    stLENS2_428[0].fEnergy := 8280.000000; stLENS2_428[0].fLow := 51.070000; stLENS2_428[0].fHigh := 10000.000000;
    stLENS2_428[1].fEnergy := 8291.222140; stLENS2_428[1].fLow := 50.858061; stLENS2_428[1].fHigh := 10000.000000;
    stLENS2_428[2].fEnergy := 8307.821178; stLENS2_428[2].fLow := 50.642862; stLENS2_428[2].fHigh := 10000.000000;
    stLENS2_428[3].fEnergy := 8324.453447; stLENS2_428[3].fLow := 50.428659; stLENS2_428[3].fHigh := 10000.000000;
    stLENS2_428[4].fEnergy := 8341.119014; stLENS2_428[4].fLow := 50.215449; stLENS2_428[4].fHigh := 10000.000000;
    stLENS2_428[5].fEnergy := 8357.817945; stLENS2_428[5].fLow := 50.003226; stLENS2_428[5].fHigh := 10000.000000;
    stLENS2_428[6].fEnergy := 8374.550308; stLENS2_428[6].fLow := 49.791984; stLENS2_428[6].fHigh := 10000.000000;
    stLENS2_428[7].fEnergy := 8391.316169; stLENS2_428[7].fLow := 49.581721; stLENS2_428[7].fHigh := 10000.000000;
    stLENS2_428[8].fEnergy := 8408.115595; stLENS2_428[8].fLow := 49.372429; stLENS2_428[8].fHigh := 10000.000000;
    stLENS2_428[9].fEnergy := 8424.948653; stLENS2_428[9].fLow := 49.164106; stLENS2_428[9].fHigh := 10000.000000;
    stLENS2_428[10].fEnergy := 8441.815412; stLENS2_428[10].fLow := 48.956745; stLENS2_428[10].fHigh := 10000.000000;
    stLENS2_428[11].fEnergy := 8458.715938; stLENS2_428[11].fLow := 48.750343; stLENS2_428[11].fHigh := 10000.000000;
    stLENS2_428[12].fEnergy := 8475.650298; stLENS2_428[12].fLow := 48.544894; stLENS2_428[12].fHigh := 10000.000000;
    stLENS2_428[13].fEnergy := 8492.618561; stLENS2_428[13].fLow := 48.340393; stLENS2_428[13].fHigh := 10000.000000;
    stLENS2_428[14].fEnergy := 8509.620795; stLENS2_428[14].fLow := 48.136837; stLENS2_428[14].fHigh := 10000.000000;
    stLENS2_428[15].fEnergy := 8526.657067; stLENS2_428[15].fLow := 47.934219; stLENS2_428[15].fHigh := 10000.000000;
    stLENS2_428[16].fEnergy := 8543.727446; stLENS2_428[16].fLow := 47.732537; stLENS2_428[16].fHigh := 10000.000000;
    stLENS2_428[17].fEnergy := 8560.832000; stLENS2_428[17].fLow := 47.531784; stLENS2_428[17].fHigh := 10000.000000;
    stLENS2_428[18].fEnergy := 8577.970797; stLENS2_428[18].fLow := 47.331957; stLENS2_428[18].fHigh := 10000.000000;
    stLENS2_428[19].fEnergy := 8595.143906; stLENS2_428[19].fLow := 47.133051; stLENS2_428[19].fHigh := 10000.000000;
    stLENS2_428[20].fEnergy := 8612.351395; stLENS2_428[20].fLow := 46.935061; stLENS2_428[20].fHigh := 10000.000000;
    stLENS2_428[21].fEnergy := 8629.593334; stLENS2_428[21].fLow := 46.737983; stLENS2_428[21].fHigh := 10000.000000;
    stLENS2_428[22].fEnergy := 8646.869792; stLENS2_428[22].fLow := 46.541812; stLENS2_428[22].fHigh := 10000.000000;
    stLENS2_428[23].fEnergy := 8664.180837; stLENS2_428[23].fLow := 46.346544; stLENS2_428[23].fHigh := 10000.000000;
    stLENS2_428[24].fEnergy := 8681.526538; stLENS2_428[24].fLow := 46.152174; stLENS2_428[24].fHigh := 10000.000000;
    stLENS2_428[25].fEnergy := 8698.906966; stLENS2_428[25].fLow := 45.958699; stLENS2_428[25].fHigh := 10000.000000;
    stLENS2_428[26].fEnergy := 8716.322189; stLENS2_428[26].fLow := 45.766112; stLENS2_428[26].fHigh := 10000.000000;
    stLENS2_428[27].fEnergy := 8733.772278; stLENS2_428[27].fLow := 45.574411; stLENS2_428[27].fHigh := 10000.000000;
    stLENS2_428[28].fEnergy := 8751.257302; stLENS2_428[28].fLow := 45.383591; stLENS2_428[28].fHigh := 10000.000000;
    stLENS2_428[29].fEnergy := 8768.777330; stLENS2_428[29].fLow := 45.193647; stLENS2_428[29].fHigh := 10000.000000;
    stLENS2_428[30].fEnergy := 8786.332434; stLENS2_428[30].fLow := 45.004575; stLENS2_428[30].fHigh := 10000.000000;
    stLENS2_428[31].fEnergy := 8803.922684; stLENS2_428[31].fLow := 44.816371; stLENS2_428[31].fHigh := 10000.000000;
    stLENS2_428[32].fEnergy := 8821.548149; stLENS2_428[32].fLow := 44.629030; stLENS2_428[32].fHigh := 10000.000000;
    stLENS2_428[33].fEnergy := 8839.208900; stLENS2_428[33].fLow := 44.442549; stLENS2_428[33].fHigh := 10000.000000;
    stLENS2_428[34].fEnergy := 8856.905008; stLENS2_428[34].fLow := 44.256922; stLENS2_428[34].fHigh := 10000.000000;
    stLENS2_428[35].fEnergy := 8874.636543; stLENS2_428[35].fLow := 44.072147; stLENS2_428[35].fHigh := 10000.000000;
    stLENS2_428[36].fEnergy := 8892.403578; stLENS2_428[36].fLow := 43.888218; stLENS2_428[36].fHigh := 10000.000000;
    stLENS2_428[37].fEnergy := 8910.206181; stLENS2_428[37].fLow := 43.705132; stLENS2_428[37].fHigh := 10000.000000;
    stLENS2_428[38].fEnergy := 8928.044426; stLENS2_428[38].fLow := 43.522884; stLENS2_428[38].fHigh := 10000.000000;
    stLENS2_428[39].fEnergy := 8945.918383; stLENS2_428[39].fLow := 43.341470; stLENS2_428[39].fHigh := 10000.000000;
    stLENS2_428[40].fEnergy := 8963.828123; stLENS2_428[40].fLow := 43.160887; stLENS2_428[40].fHigh := 10000.000000;
    stLENS2_428[41].fEnergy := 8981.773719; stLENS2_428[41].fLow := 42.981129; stLENS2_428[41].fHigh := 10000.000000;
    stLENS2_428[42].fEnergy := 8999.755242; stLENS2_428[42].fLow := 42.802194; stLENS2_428[42].fHigh := 10000.000000;
    stLENS2_428[43].fEnergy := 9017.772764; stLENS2_428[43].fLow := 42.624076; stLENS2_428[43].fHigh := 10000.000000;
    stLENS2_428[44].fEnergy := 9035.826357; stLENS2_428[44].fLow := 42.446773; stLENS2_428[44].fHigh := 10000.000000;
    stLENS2_428[45].fEnergy := 9053.916094; stLENS2_428[45].fLow := 42.270279; stLENS2_428[45].fHigh := 10000.000000;
    stLENS2_428[46].fEnergy := 9072.042046; stLENS2_428[46].fLow := 42.094591; stLENS2_428[46].fHigh := 10000.000000;
    stLENS2_428[47].fEnergy := 9090.204286; stLENS2_428[47].fLow := 41.919706; stLENS2_428[47].fHigh := 10000.000000;
    stLENS2_428[48].fEnergy := 9108.402887; stLENS2_428[48].fLow := 41.745618; stLENS2_428[48].fHigh := 10000.000000;
    stLENS2_428[49].fEnergy := 9126.637922; stLENS2_428[49].fLow := 41.572325; stLENS2_428[49].fHigh := 10000.000000;
    stLENS2_428[50].fEnergy := 9144.909463; stLENS2_428[50].fLow := 41.399822; stLENS2_428[50].fHigh := 10000.000000;
    stLENS2_428[51].fEnergy := 9163.217584; stLENS2_428[51].fLow := 41.228106; stLENS2_428[51].fHigh := 10000.000000;
    stLENS2_428[52].fEnergy := 9181.562358; stLENS2_428[52].fLow := 41.057172; stLENS2_428[52].fHigh := 10000.000000;
    stLENS2_428[53].fEnergy := 9199.943858; stLENS2_428[53].fLow := 40.887017; stLENS2_428[53].fHigh := 10000.000000;
    stLENS2_428[54].fEnergy := 9218.362158; stLENS2_428[54].fLow := 40.717637; stLENS2_428[54].fHigh := 10000.000000;
    stLENS2_428[55].fEnergy := 9236.817331; stLENS2_428[55].fLow := 40.549028; stLENS2_428[55].fHigh := 10000.000000;
    stLENS2_428[56].fEnergy := 9255.309452; stLENS2_428[56].fLow := 40.381186; stLENS2_428[56].fHigh := 10000.000000;
    stLENS2_428[57].fEnergy := 9273.838594; stLENS2_428[57].fLow := 40.214108; stLENS2_428[57].fHigh := 10000.000000;
    stLENS2_428[58].fEnergy := 9292.404831; stLENS2_428[58].fLow := 40.047790; stLENS2_428[58].fHigh := 10000.000000;
    stLENS2_428[59].fEnergy := 9311.008238; stLENS2_428[59].fLow := 39.882228; stLENS2_428[59].fHigh := 10000.000000;
    stLENS2_428[60].fEnergy := 9329.648889; stLENS2_428[60].fLow := 39.717419; stLENS2_428[60].fHigh := 10000.000000;
    stLENS2_428[61].fEnergy := 9348.326858; stLENS2_428[61].fLow := 39.553358; stLENS2_428[61].fHigh := 10000.000000;
    stLENS2_428[62].fEnergy := 9367.042221; stLENS2_428[62].fLow := 39.390043; stLENS2_428[62].fHigh := 10000.000000;
    stLENS2_428[63].fEnergy := 9385.795052; stLENS2_428[63].fLow := 39.227469; stLENS2_428[63].fHigh := 10000.000000;
    stLENS2_428[64].fEnergy := 9404.585426; stLENS2_428[64].fLow := 39.065634; stLENS2_428[64].fHigh := 10000.000000;
    stLENS2_428[65].fEnergy := 9423.413419; stLENS2_428[65].fLow := 38.904532; stLENS2_428[65].fHigh := 10000.000000;
    stLENS2_428[66].fEnergy := 9442.279105; stLENS2_428[66].fLow := 38.744161; stLENS2_428[66].fHigh := 10000.000000;
    stLENS2_428[67].fEnergy := 9461.182561; stLENS2_428[67].fLow := 38.584518; stLENS2_428[67].fHigh := 10000.000000;
    stLENS2_428[68].fEnergy := 9480.123861; stLENS2_428[68].fLow := 38.425598; stLENS2_428[68].fHigh := 10000.000000;
    stLENS2_428[69].fEnergy := 9499.103081; stLENS2_428[69].fLow := 38.267398; stLENS2_428[69].fHigh := 10000.000000;
    stLENS2_428[70].fEnergy := 9518.120298; stLENS2_428[70].fLow := 38.109915; stLENS2_428[70].fHigh := 10000.000000;
    stLENS2_428[71].fEnergy := 9537.175588; stLENS2_428[71].fLow := 37.953145; stLENS2_428[71].fHigh := 10000.000000;
    stLENS2_428[72].fEnergy := 9556.269026; stLENS2_428[72].fLow := 37.797085; stLENS2_428[72].fHigh := 10000.000000;
    stLENS2_428[73].fEnergy := 9575.400690; stLENS2_428[73].fLow := 37.641731; stLENS2_428[73].fHigh := 10000.000000;
    stLENS2_428[74].fEnergy := 9594.570654; stLENS2_428[74].fLow := 37.487079; stLENS2_428[74].fHigh := 10000.000000;
    stLENS2_428[75].fEnergy := 9613.778998; stLENS2_428[75].fLow := 37.333127; stLENS2_428[75].fHigh := 10000.000000;
    stLENS2_428[76].fEnergy := 9633.025796; stLENS2_428[76].fLow := 37.179871; stLENS2_428[76].fHigh := 10000.000000;
    stLENS2_428[77].fEnergy := 9652.311127; stLENS2_428[77].fLow := 37.027308; stLENS2_428[77].fHigh := 10000.000000;
    stLENS2_428[78].fEnergy := 9671.635066; stLENS2_428[78].fLow := 36.875434; stLENS2_428[78].fHigh := 10000.000000;
    stLENS2_428[79].fEnergy := 9690.997693; stLENS2_428[79].fLow := 36.724245; stLENS2_428[79].fHigh := 10000.000000;
    stLENS2_428[80].fEnergy := 9710.399083; stLENS2_428[80].fLow := 36.573740; stLENS2_428[80].fHigh := 10000.000000;
    stLENS2_428[81].fEnergy := 9729.839315; stLENS2_428[81].fLow := 36.423913; stLENS2_428[81].fHigh := 10000.000000;
    stLENS2_428[82].fEnergy := 9749.318466; stLENS2_428[82].fLow := 36.274762; stLENS2_428[82].fHigh := 10000.000000;
    stLENS2_428[83].fEnergy := 9768.836615; stLENS2_428[83].fLow := 36.126284; stLENS2_428[83].fHigh := 10000.000000;
    stLENS2_428[84].fEnergy := 9788.393839; stLENS2_428[84].fLow := 35.978476; stLENS2_428[84].fHigh := 10000.000000;
    stLENS2_428[85].fEnergy := 9807.990216; stLENS2_428[85].fLow := 35.831333; stLENS2_428[85].fHigh := 10000.000000;
    stLENS2_428[86].fEnergy := 9827.625826; stLENS2_428[86].fLow := 35.684854; stLENS2_428[86].fHigh := 10000.000000;
    stLENS2_428[87].fEnergy := 9847.300746; stLENS2_428[87].fLow := 35.539034; stLENS2_428[87].fHigh := 10000.000000;
    stLENS2_428[88].fEnergy := 9867.015055; stLENS2_428[88].fLow := 35.393871; stLENS2_428[88].fHigh := 10000.000000;
    stLENS2_428[89].fEnergy := 9886.768832; stLENS2_428[89].fLow := 35.249361; stLENS2_428[89].fHigh := 10000.000000;
    stLENS2_428[90].fEnergy := 9906.562157; stLENS2_428[90].fLow := 35.105501; stLENS2_428[90].fHigh := 10000.000000;
    stLENS2_428[91].fEnergy := 9926.395107; stLENS2_428[91].fLow := 34.962289; stLENS2_428[91].fHigh := 10000.000000;
    stLENS2_428[92].fEnergy := 9946.267764; stLENS2_428[92].fLow := 34.819720; stLENS2_428[92].fHigh := 10000.000000;
    stLENS2_428[93].fEnergy := 9966.180205; stLENS2_428[93].fLow := 34.677792; stLENS2_428[93].fHigh := 10000.000000;
    stLENS2_428[94].fEnergy := 9986.132511; stLENS2_428[94].fLow := 34.536501; stLENS2_428[94].fHigh := 10000.000000;
    stLENS2_428[95].fEnergy := 10006.124762; stLENS2_428[95].fLow := 34.395846; stLENS2_428[95].fHigh := 10000.000000;
    stLENS2_428[96].fEnergy := 10026.157037; stLENS2_428[96].fLow := 34.255822; stLENS2_428[96].fHigh := 10000.000000;
    stLENS2_428[97].fEnergy := 10046.229416; stLENS2_428[97].fLow := 34.116426; stLENS2_428[97].fHigh := 3540.238801;
    stLENS2_428[98].fEnergy := 10066.341981; stLENS2_428[98].fLow := 33.977656; stLENS2_428[98].fHigh := 2735.412827;
    stLENS2_428[99].fEnergy := 10086.494811; stLENS2_428[99].fLow := 33.839508; stLENS2_428[99].fHigh := 2113.553282;
    stLENS2_428[100].fEnergy := 10106.687987; stLENS2_428[100].fLow := 33.701980; stLENS2_428[100].fHigh := 1633.065192;
    stLENS2_428[101].fEnergy := 10126.921590; stLENS2_428[101].fLow := 33.565068; stLENS2_428[101].fHigh := 1261.809648;
    stLENS2_428[102].fEnergy := 10147.195701; stLENS2_428[102].fLow := 33.428769; stLENS2_428[102].fHigh := 993.711493;
    stLENS2_428[103].fEnergy := 10167.510400; stLENS2_428[103].fLow := 33.293081; stLENS2_428[103].fHigh := 931.972333;
    stLENS2_428[104].fEnergy := 10187.865769; stLENS2_428[104].fLow := 33.158001; stLENS2_428[104].fHigh := 874.069019;
    stLENS2_428[105].fEnergy := 10208.261890; stLENS2_428[105].fLow := 33.023525; stLENS2_428[105].fHigh := 819.763230;
    stLENS2_428[106].fEnergy := 10228.698844; stLENS2_428[106].fLow := 32.889652; stLENS2_428[106].fHigh := 768.831452;
    stLENS2_428[107].fEnergy := 10249.176713; stLENS2_428[107].fLow := 32.756377; stLENS2_428[107].fHigh := 721.064059;
    stLENS2_428[108].fEnergy := 10269.695578; stLENS2_428[108].fLow := 32.623697; stLENS2_428[108].fHigh := 676.264447;
    stLENS2_428[109].fEnergy := 10290.255523; stLENS2_428[109].fLow := 32.491611; stLENS2_428[109].fHigh := 634.248229;
    stLENS2_428[110].fEnergy := 10310.856628; stLENS2_428[110].fLow := 32.360116; stLENS2_428[110].fHigh := 594.842473;
    stLENS2_428[111].fEnergy := 10331.498977; stLENS2_428[111].fLow := 32.229207; stLENS2_428[111].fHigh := 557.884991;
    stLENS2_428[112].fEnergy := 10352.182651; stLENS2_428[112].fLow := 32.098884; stLENS2_428[112].fHigh := 523.223673;
    stLENS2_428[113].fEnergy := 10372.907735; stLENS2_428[113].fLow := 31.969142; stLENS2_428[113].fHigh := 490.715857;
    stLENS2_428[114].fEnergy := 10393.674310; stLENS2_428[114].fLow := 31.839978; stLENS2_428[114].fHigh := 460.227748;
    stLENS2_428[115].fEnergy := 10414.482460; stLENS2_428[115].fLow := 31.711392; stLENS2_428[115].fHigh := 431.633861;
    stLENS2_428[116].fEnergy := 10435.332268; stLENS2_428[116].fLow := 31.583378; stLENS2_428[116].fHigh := 404.816508;
    stLENS2_428[117].fEnergy := 10456.223817; stLENS2_428[117].fLow := 31.455935; stLENS2_428[117].fHigh := 379.665313;
    stLENS2_428[118].fEnergy := 10477.157191; stLENS2_428[118].fLow := 31.329061; stLENS2_428[118].fHigh := 356.076759;
    stLENS2_428[119].fEnergy := 10498.132473; stLENS2_428[119].fLow := 31.202751; stLENS2_428[119].fHigh := 333.953758;
    stLENS2_428[120].fEnergy := 10519.149749; stLENS2_428[120].fLow := 31.077004; stLENS2_428[120].fHigh := 315.209076;
    stLENS2_428[121].fEnergy := 10540.209100; stLENS2_428[121].fLow := 30.951817; stLENS2_428[121].fHigh := 308.488005;
    stLENS2_428[122].fEnergy := 10561.310613; stLENS2_428[122].fLow := 30.827186; stLENS2_428[122].fHigh := 301.910244;
    stLENS2_428[123].fEnergy := 10582.454371; stLENS2_428[123].fLow := 30.703111; stLENS2_428[123].fHigh := 295.472738;
    stLENS2_428[124].fEnergy := 10603.640459; stLENS2_428[124].fLow := 30.579587; stLENS2_428[124].fHigh := 289.172496;
    stLENS2_428[125].fEnergy := 10624.868961; stLENS2_428[125].fLow := 30.456612; stLENS2_428[125].fHigh := 283.006591;
    stLENS2_428[126].fEnergy := 10646.139963; stLENS2_428[126].fLow := 30.334184; stLENS2_428[126].fHigh := 276.972160;
    stLENS2_428[127].fEnergy := 10667.453549; stLENS2_428[127].fLow := 30.212299; stLENS2_428[127].fHigh := 271.066398;
    stLENS2_428[128].fEnergy := 10688.809806; stLENS2_428[128].fLow := 30.090956; stLENS2_428[128].fHigh := 265.286563;
    stLENS2_428[129].fEnergy := 10710.208817; stLENS2_428[129].fLow := 29.970152; stLENS2_428[129].fHigh := 259.629968;
    stLENS2_428[130].fEnergy := 10731.650669; stLENS2_428[130].fLow := 29.849884; stLENS2_428[130].fHigh := 254.093987;
    stLENS2_428[131].fEnergy := 10753.135448; stLENS2_428[131].fLow := 29.730149; stLENS2_428[131].fHigh := 248.676047;
    stLENS2_428[132].fEnergy := 10774.663240; stLENS2_428[132].fLow := 29.610945; stLENS2_428[132].fHigh := 243.373631;
    stLENS2_428[133].fEnergy := 10796.234130; stLENS2_428[133].fLow := 29.492270; stLENS2_428[133].fHigh := 238.184277;
    stLENS2_428[134].fEnergy := 10817.848205; stLENS2_428[134].fLow := 29.374121; stLENS2_428[134].fHigh := 233.105573;
    stLENS2_428[135].fEnergy := 10839.505552; stLENS2_428[135].fLow := 29.256495; stLENS2_428[135].fHigh := 228.135160;
    stLENS2_428[136].fEnergy := 10861.206256; stLENS2_428[136].fLow := 29.139391; stLENS2_428[136].fHigh := 223.270729;
    stLENS2_428[137].fEnergy := 10882.950406; stLENS2_428[137].fLow := 29.022804; stLENS2_428[137].fHigh := 218.510021;
    stLENS2_428[138].fEnergy := 10904.738087; stLENS2_428[138].fLow := 28.906734; stLENS2_428[138].fHigh := 213.850823;
    stLENS2_428[139].fEnergy := 10926.569387; stLENS2_428[139].fLow := 28.791177; stLENS2_428[139].fHigh := 209.290971;
    stLENS2_428[140].fEnergy := 10948.444394; stLENS2_428[140].fLow := 28.676132; stLENS2_428[140].fHigh := 204.828347;
    stLENS2_428[141].fEnergy := 10970.363194; stLENS2_428[141].fLow := 28.561595; stLENS2_428[141].fHigh := 200.460878;
    stLENS2_428[142].fEnergy := 10992.325876; stLENS2_428[142].fLow := 28.447564; stLENS2_428[142].fHigh := 196.186534;
    stLENS2_428[143].fEnergy := 11014.332527; stLENS2_428[143].fLow := 28.334037; stLENS2_428[143].fHigh := 192.003330;
    stLENS2_428[144].fEnergy := 11036.383235; stLENS2_428[144].fLow := 28.221011; stLENS2_428[144].fHigh := 187.909324;
    stLENS2_428[145].fEnergy := 11058.478089; stLENS2_428[145].fLow := 28.108485; stLENS2_428[145].fHigh := 183.902611;
    stLENS2_428[146].fEnergy := 11080.617177; stLENS2_428[146].fLow := 27.996455; stLENS2_428[146].fHigh := 179.981333;
    stLENS2_428[147].fEnergy := 11102.800587; stLENS2_428[147].fLow := 27.884919; stLENS2_428[147].fHigh := 177.021145;
    stLENS2_428[148].fEnergy := 11125.028409; stLENS2_428[148].fLow := 27.773876; stLENS2_428[148].fHigh := 175.207335;
    stLENS2_428[149].fEnergy := 11147.300731; stLENS2_428[149].fLow := 27.663322; stLENS2_428[149].fHigh := 173.412110;
    stLENS2_428[150].fEnergy := 11169.617642; stLENS2_428[150].fLow := 27.553255; stLENS2_428[150].fHigh := 171.635280;
    stLENS2_428[151].fEnergy := 11191.979231; stLENS2_428[151].fLow := 27.443673; stLENS2_428[151].fHigh := 169.876655;
    stLENS2_428[152].fEnergy := 11214.385588; stLENS2_428[152].fLow := 27.334574; stLENS2_428[152].fHigh := 168.136050;
    stLENS2_428[153].fEnergy := 11236.836803; stLENS2_428[153].fLow := 27.225955; stLENS2_428[153].fHigh := 166.413279;
    stLENS2_428[154].fEnergy := 11259.332966; stLENS2_428[154].fLow := 27.117815; stLENS2_428[154].fHigh := 164.708161;
    stLENS2_428[155].fEnergy := 11281.874165; stLENS2_428[155].fLow := 27.010150; stLENS2_428[155].fHigh := 163.020514;
    stLENS2_428[156].fEnergy := 11304.460492; stLENS2_428[156].fLow := 26.902958; stLENS2_428[156].fHigh := 161.350158;
    stLENS2_428[157].fEnergy := 11327.092037; stLENS2_428[157].fLow := 26.796238; stLENS2_428[157].fHigh := 159.696918;
    stLENS2_428[158].fEnergy := 11349.768891; stLENS2_428[158].fLow := 26.689988; stLENS2_428[158].fHigh := 158.060617;
    stLENS2_428[159].fEnergy := 11372.491143; stLENS2_428[159].fLow := 26.584204; stLENS2_428[159].fHigh := 156.441083;
    stLENS2_428[160].fEnergy := 11395.258886; stLENS2_428[160].fLow := 26.478884; stLENS2_428[160].fHigh := 154.838142;
    stLENS2_428[161].fEnergy := 11418.072209; stLENS2_428[161].fLow := 26.374027; stLENS2_428[161].fHigh := 153.251626;
    stLENS2_428[162].fEnergy := 11440.931205; stLENS2_428[162].fLow := 26.269630; stLENS2_428[162].fHigh := 151.681365;
    stLENS2_428[163].fEnergy := 11463.835964; stLENS2_428[163].fLow := 26.165692; stLENS2_428[163].fHigh := 150.127194;
    stLENS2_428[164].fEnergy := 11486.786579; stLENS2_428[164].fLow := 26.062209; stLENS2_428[164].fHigh := 148.588948;
    stLENS2_428[165].fEnergy := 11509.783141; stLENS2_428[165].fLow := 25.959180; stLENS2_428[165].fHigh := 147.066463;
    stLENS2_428[166].fEnergy := 11532.825743; stLENS2_428[166].fLow := 25.856603; stLENS2_428[166].fHigh := 145.559577;
    stLENS2_428[167].fEnergy := 11555.914475; stLENS2_428[167].fLow := 25.754475; stLENS2_428[167].fHigh := 144.068132;
    stLENS2_428[168].fEnergy := 11579.049431; stLENS2_428[168].fLow := 25.652794; stLENS2_428[168].fHigh := 142.591968;
    stLENS2_428[169].fEnergy := 11602.230704; stLENS2_428[169].fLow := 25.551559; stLENS2_428[169].fHigh := 141.130930;
    stLENS2_428[170].fEnergy := 11625.458385; stLENS2_428[170].fLow := 25.450767; stLENS2_428[170].fHigh := 139.684861;
    stLENS2_428[171].fEnergy := 11648.732568; stLENS2_428[171].fLow := 25.350416; stLENS2_428[171].fHigh := 138.253610;
    stLENS2_428[172].fEnergy := 11672.053346; stLENS2_428[172].fLow := 25.250503; stLENS2_428[172].fHigh := 136.837024;
    stLENS2_428[173].fEnergy := 11695.420813; stLENS2_428[173].fLow := 25.151028; stLENS2_428[173].fHigh := 135.434952;
    stLENS2_428[174].fEnergy := 11718.835061; stLENS2_428[174].fLow := 25.051987; stLENS2_428[174].fHigh := 134.047246;
    stLENS2_428[175].fEnergy := 11742.296184; stLENS2_428[175].fLow := 24.953380; stLENS2_428[175].fHigh := 132.673760;
    stLENS2_428[176].fEnergy := 11765.804277; stLENS2_428[176].fLow := 24.855203; stLENS2_428[176].fHigh := 131.314346;
    stLENS2_428[177].fEnergy := 11789.359433; stLENS2_428[177].fLow := 24.757454; stLENS2_428[177].fHigh := 129.968861;
    stLENS2_428[178].fEnergy := 11812.961746; stLENS2_428[178].fLow := 24.660133; stLENS2_428[178].fHigh := 128.637163;
    stLENS2_428[179].fEnergy := 11836.611311; stLENS2_428[179].fLow := 24.563236; stLENS2_428[179].fHigh := 127.319109;
    stLENS2_428[180].fEnergy := 11860.308223; stLENS2_428[180].fLow := 24.466761; stLENS2_428[180].fHigh := 126.014561;
    stLENS2_428[181].fEnergy := 11884.052576; stLENS2_428[181].fLow := 24.370708; stLENS2_428[181].fHigh := 124.723379;
    stLENS2_428[182].fEnergy := 11907.844465; stLENS2_428[182].fLow := 24.275073; stLENS2_428[182].fHigh := 123.445428;
    stLENS2_428[183].fEnergy := 11931.683985; stLENS2_428[183].fLow := 24.179854; stLENS2_428[183].fHigh := 122.180570;
    stLENS2_428[184].fEnergy := 11955.571233; stLENS2_428[184].fLow := 24.085051; stLENS2_428[184].fHigh := 120.928673;
    stLENS2_428[185].fEnergy := 11979.506302; stLENS2_428[185].fLow := 23.990660; stLENS2_428[185].fHigh := 119.689603;
    stLENS2_428[186].fEnergy := 12003.489290; stLENS2_428[186].fLow := 23.896680; stLENS2_428[186].fHigh := 118.463228;
    stLENS2_428[187].fEnergy := 12027.520291; stLENS2_428[187].fLow := 23.803109; stLENS2_428[187].fHigh := 117.249420;
    stLENS2_428[188].fEnergy := 12051.599403; stLENS2_428[188].fLow := 23.709946; stLENS2_428[188].fHigh := 116.048049;
    stLENS2_428[189].fEnergy := 12075.726721; stLENS2_428[189].fLow := 23.617187; stLENS2_428[189].fHigh := 114.858987;
    stLENS2_428[190].fEnergy := 12099.902342; stLENS2_428[190].fLow := 23.524831; stLENS2_428[190].fHigh := 113.682108;
    stLENS2_428[191].fEnergy := 12124.126363; stLENS2_428[191].fLow := 23.432877; stLENS2_428[191].fHigh := 112.517289;
    stLENS2_428[192].fEnergy := 12148.398880; stLENS2_428[192].fLow := 23.341322; stLENS2_428[192].fHigh := 111.364404;
    stLENS2_428[193].fEnergy := 12172.719991; stLENS2_428[193].fLow := 23.250165; stLENS2_428[193].fHigh := 110.223332;
    stLENS2_428[194].fEnergy := 12197.089792; stLENS2_428[194].fLow := 23.159404; stLENS2_428[194].fHigh := 109.093952;
    stLENS2_428[195].fEnergy := 12221.508382; stLENS2_428[195].fLow := 23.069036; stLENS2_428[195].fHigh := 107.976144;
    stLENS2_428[196].fEnergy := 12245.975858; stLENS2_428[196].fLow := 22.979060; stLENS2_428[196].fHigh := 106.869789;
    stLENS2_428[197].fEnergy := 12270.492318; stLENS2_428[197].fLow := 22.889475; stLENS2_428[197].fHigh := 105.774771;
    stLENS2_428[198].fEnergy := 12295.057860; stLENS2_428[198].fLow := 22.800277; stLENS2_428[198].fHigh := 104.690972;
    stLENS2_428[199].fEnergy := 12319.672583; stLENS2_428[199].fLow := 22.711467; stLENS2_428[199].fHigh := 103.618278;
    stLENS2_428[200].fEnergy := 12344.336584; stLENS2_428[200].fLow := 22.623041; stLENS2_428[200].fHigh := 102.556575;
    stLENS2_428[201].fEnergy := 12369.049962; stLENS2_428[201].fLow := 22.534998; stLENS2_428[201].fHigh := 101.505751;
    stLENS2_428[202].fEnergy := 12393.812816; stLENS2_428[202].fLow := 22.447336; stLENS2_428[202].fHigh := 100.465694;
    stLENS2_428[203].fEnergy := 12418.625246; stLENS2_428[203].fLow := 22.360053; stLENS2_428[203].fHigh := 99.648563;
    stLENS2_428[204].fEnergy := 12443.487350; stLENS2_428[204].fLow := 22.273148; stLENS2_428[204].fHigh := 99.011458;
    stLENS2_428[205].fEnergy := 12468.399229; stLENS2_428[205].fLow := 22.186619; stLENS2_428[205].fHigh := 98.378425;
    stLENS2_428[206].fEnergy := 12493.360981; stLENS2_428[206].fLow := 22.100463; stLENS2_428[206].fHigh := 97.749441;
    stLENS2_428[207].fEnergy := 12518.372706; stLENS2_428[207].fLow := 22.014680; stLENS2_428[207].fHigh := 97.124477;
    stLENS2_428[208].fEnergy := 12543.434505; stLENS2_428[208].fLow := 21.929268; stLENS2_428[208].fHigh := 96.503509;
    stLENS2_428[209].fEnergy := 12568.546477; stLENS2_428[209].fLow := 21.844224; stLENS2_428[209].fHigh := 95.886512;
    stLENS2_428[210].fEnergy := 12593.708724; stLENS2_428[210].fLow := 21.759547; stLENS2_428[210].fHigh := 95.273459;
    stLENS2_428[211].fEnergy := 12618.921346; stLENS2_428[211].fLow := 21.675236; stLENS2_428[211].fHigh := 94.664326;
    stLENS2_428[212].fEnergy := 12644.184443; stLENS2_428[212].fLow := 21.591289; stLENS2_428[212].fHigh := 94.059087;
    stLENS2_428[213].fEnergy := 12669.498117; stLENS2_428[213].fLow := 21.507703; stLENS2_428[213].fHigh := 93.457718;
    stLENS2_428[214].fEnergy := 12694.862470; stLENS2_428[214].fLow := 21.424478; stLENS2_428[214].fHigh := 92.860194;
    stLENS2_428[215].fEnergy := 12720.277601; stLENS2_428[215].fLow := 21.341611; stLENS2_428[215].fHigh := 92.266490;
    stLENS2_428[216].fEnergy := 12745.743614; stLENS2_428[216].fLow := 21.259102; stLENS2_428[216].fHigh := 91.676582;
    stLENS2_428[217].fEnergy := 12771.260610; stLENS2_428[217].fLow := 21.176947; stLENS2_428[217].fHigh := 91.090445;
    stLENS2_428[218].fEnergy := 12796.828690; stLENS2_428[218].fLow := 21.095147; stLENS2_428[218].fHigh := 90.508056;
    stLENS2_428[219].fEnergy := 12822.447958; stLENS2_428[219].fLow := 21.013698; stLENS2_428[219].fHigh := 89.929391;
    stLENS2_428[220].fEnergy := 12848.118516; stLENS2_428[220].fLow := 20.932599; stLENS2_428[220].fHigh := 89.354425;
    stLENS2_428[221].fEnergy := 12873.840467; stLENS2_428[221].fLow := 20.851850; stLENS2_428[221].fHigh := 88.783135;
    stLENS2_428[222].fEnergy := 12899.613913; stLENS2_428[222].fLow := 20.771447; stLENS2_428[222].fHigh := 88.215498;
    stLENS2_428[223].fEnergy := 12925.438957; stLENS2_428[223].fLow := 20.691390; stLENS2_428[223].fHigh := 87.651490;
    stLENS2_428[224].fEnergy := 12951.315703; stLENS2_428[224].fLow := 20.611677; stLENS2_428[224].fHigh := 87.091088;
    stLENS2_428[225].fEnergy := 12977.244254; stLENS2_428[225].fLow := 20.532306; stLENS2_428[225].fHigh := 86.534269;
    stLENS2_428[226].fEnergy := 13003.224714; stLENS2_428[226].fLow := 20.453276; stLENS2_428[226].fHigh := 85.981010;
    stLENS2_428[227].fEnergy := 13029.257188; stLENS2_428[227].fLow := 20.374584; stLENS2_428[227].fHigh := 85.431289;
    stLENS2_428[228].fEnergy := 13055.341778; stLENS2_428[228].fLow := 20.296231; stLENS2_428[228].fHigh := 84.885081;
    stLENS2_428[229].fEnergy := 13081.478590; stLENS2_428[229].fLow := 20.218213; stLENS2_428[229].fHigh := 84.342367;
    stLENS2_428[230].fEnergy := 13107.667727; stLENS2_428[230].fLow := 20.140530; stLENS2_428[230].fHigh := 83.803122;
    stLENS2_428[231].fEnergy := 13133.909296; stLENS2_428[231].fLow := 20.063179; stLENS2_428[231].fHigh := 83.267324;
    stLENS2_428[232].fEnergy := 13160.203399; stLENS2_428[232].fLow := 19.986160; stLENS2_428[232].fHigh := 82.734953;
    stLENS2_428[233].fEnergy := 13186.550144; stLENS2_428[233].fLow := 19.909471; stLENS2_428[233].fHigh := 82.205985;
    stLENS2_428[234].fEnergy := 13212.949635; stLENS2_428[234].fLow := 19.833110; stLENS2_428[234].fHigh := 81.680399;
    stLENS2_428[235].fEnergy := 13239.401978; stLENS2_428[235].fLow := 19.757076; stLENS2_428[235].fHigh := 81.158173;
    stLENS2_428[236].fEnergy := 13265.907278; stLENS2_428[236].fLow := 19.681367; stLENS2_428[236].fHigh := 80.639286;
    stLENS2_428[237].fEnergy := 13292.465642; stLENS2_428[237].fLow := 19.605981; stLENS2_428[237].fHigh := 80.123717;
    stLENS2_428[238].fEnergy := 13319.077176; stLENS2_428[238].fLow := 19.530918; stLENS2_428[238].fHigh := 79.611444;
    stLENS2_428[239].fEnergy := 13345.741987; stLENS2_428[239].fLow := 19.456176; stLENS2_428[239].fHigh := 79.102446;
    stLENS2_428[240].fEnergy := 13372.460180; stLENS2_428[240].fLow := 19.381752; stLENS2_428[240].fHigh := 78.596703;
    stLENS2_428[241].fEnergy := 13399.231863; stLENS2_428[241].fLow := 19.307647; stLENS2_428[241].fHigh := 78.094193;
    stLENS2_428[242].fEnergy := 13426.057143; stLENS2_428[242].fLow := 19.233858; stLENS2_428[242].fHigh := 77.594896;
    stLENS2_428[243].fEnergy := 13452.936127; stLENS2_428[243].fLow := 19.160383; stLENS2_428[243].fHigh := 77.098791;
    stLENS2_428[244].fEnergy := 13479.868924; stLENS2_428[244].fLow := 19.087223; stLENS2_428[244].fHigh := 76.605858;
    stLENS2_428[245].fEnergy := 13506.855639; stLENS2_428[245].fLow := 19.014374; stLENS2_428[245].fHigh := 76.116076;
    stLENS2_428[246].fEnergy := 13533.896382; stLENS2_428[246].fLow := 18.941835; stLENS2_428[246].fHigh := 75.629426;
    stLENS2_428[247].fEnergy := 13560.991261; stLENS2_428[247].fLow := 18.869606; stLENS2_428[247].fHigh := 75.145888;
    stLENS2_428[248].fEnergy := 13588.140383; stLENS2_428[248].fLow := 18.797684; stLENS2_428[248].fHigh := 74.665441;
    stLENS2_428[249].fEnergy := 13615.343858; stLENS2_428[249].fLow := 18.726068; stLENS2_428[249].fHigh := 74.188065;
    stLENS2_428[250].fEnergy := 13642.601795; stLENS2_428[250].fLow := 18.654758; stLENS2_428[250].fHigh := 73.713742;
    stLENS2_428[251].fEnergy := 13669.914302; stLENS2_428[251].fLow := 18.583750; stLENS2_428[251].fHigh := 73.242452;
    stLENS2_428[252].fEnergy := 13697.281489; stLENS2_428[252].fLow := 18.513045; stLENS2_428[252].fHigh := 72.774174;
    stLENS2_428[253].fEnergy := 13724.703465; stLENS2_428[253].fLow := 18.442640; stLENS2_428[253].fHigh := 72.308891;
    stLENS2_428[254].fEnergy := 13752.180339; stLENS2_428[254].fLow := 18.372535; stLENS2_428[254].fHigh := 71.846582;
    stLENS2_428[255].fEnergy := 13779.712223; stLENS2_428[255].fLow := 18.302727; stLENS2_428[255].fHigh := 71.387229;
    stLENS2_428[256].fEnergy := 13807.299225; stLENS2_428[256].fLow := 18.233216; stLENS2_428[256].fHigh := 70.930813;
    stLENS2_428[257].fEnergy := 13834.941456; stLENS2_428[257].fLow := 18.164000; stLENS2_428[257].fHigh := 70.477315;
    stLENS2_428[258].fEnergy := 13862.639028; stLENS2_428[258].fLow := 18.095078; stLENS2_428[258].fHigh := 70.026717;
    stLENS2_428[259].fEnergy := 13890.392049; stLENS2_428[259].fLow := 18.026448; stLENS2_428[259].fHigh := 69.578999;
    stLENS2_428[260].fEnergy := 13918.200633; stLENS2_428[260].fLow := 17.958109; stLENS2_428[260].fHigh := 69.134144;
    stLENS2_428[261].fEnergy := 13946.064889; stLENS2_428[261].fLow := 17.890060; stLENS2_428[261].fHigh := 68.692133;
    stLENS2_428[262].fEnergy := 13973.984929; stLENS2_428[262].fLow := 17.822299; stLENS2_428[262].fHigh := 68.252948;
    stLENS2_428[263].fEnergy := 14001.960866; stLENS2_428[263].fLow := 17.754826; stLENS2_428[263].fHigh := 67.816572;
    stLENS2_428[264].fEnergy := 14029.992810; stLENS2_428[264].fLow := 17.687638; stLENS2_428[264].fHigh := 67.382985;
    stLENS2_428[265].fEnergy := 14058.080875; stLENS2_428[265].fLow := 17.787537; stLENS2_428[265].fHigh := 66.952170;
    stLENS2_428[266].fEnergy := 14086.225171; stLENS2_428[266].fLow := 17.721177; stLENS2_428[266].fHigh := 66.524110;
    stLENS2_428[267].fEnergy := 14114.425813; stLENS2_428[267].fLow := 17.655064; stLENS2_428[267].fHigh := 66.098786;
    stLENS2_428[268].fEnergy := 14142.682912; stLENS2_428[268].fLow := 17.589198; stLENS2_428[268].fHigh := 65.676182;
    stLENS2_428[269].fEnergy := 14170.996582; stLENS2_428[269].fLow := 17.523578; stLENS2_428[269].fHigh := 65.256279;
    stLENS2_428[270].fEnergy := 14199.366936; stLENS2_428[270].fLow := 17.458202; stLENS2_428[270].fHigh := 64.839062;
    stLENS2_428[271].fEnergy := 14227.794088; stLENS2_428[271].fLow := 17.393071; stLENS2_428[271].fHigh := 64.424512;
    stLENS2_428[272].fEnergy := 14256.278151; stLENS2_428[272].fLow := 17.328182; stLENS2_428[272].fHigh := 64.012612;
    stLENS2_428[273].fEnergy := 14284.819238; stLENS2_428[273].fLow := 17.263536; stLENS2_428[273].fHigh := 63.603346;
    stLENS2_428[274].fEnergy := 14313.417466; stLENS2_428[274].fLow := 17.199130; stLENS2_428[274].fHigh := 63.196696;
    stLENS2_428[275].fEnergy := 14342.072946; stLENS2_428[275].fLow := 17.134965; stLENS2_428[275].fHigh := 62.792647;
    stLENS2_428[276].fEnergy := 14370.785796; stLENS2_428[276].fLow := 17.071039; stLENS2_428[276].fHigh := 62.391180;
    stLENS2_428[277].fEnergy := 14399.556128; stLENS2_428[277].fLow := 17.007352; stLENS2_428[277].fHigh := 61.992281;
    stLENS2_428[278].fEnergy := 14428.384059; stLENS2_428[278].fLow := 16.943903; stLENS2_428[278].fHigh := 61.595932;
    stLENS2_428[279].fEnergy := 14457.269703; stLENS2_428[279].fLow := 16.880690; stLENS2_428[279].fHigh := 61.202116;
    stLENS2_428[280].fEnergy := 14486.213176; stLENS2_428[280].fLow := 16.817713; stLENS2_428[280].fHigh := 60.810819;
    stLENS2_428[281].fEnergy := 14515.214594; stLENS2_428[281].fLow := 16.754971; stLENS2_428[281].fHigh := 60.422024;
    stLENS2_428[282].fEnergy := 14544.274073; stLENS2_428[282].fLow := 16.692463; stLENS2_428[282].fHigh := 60.035714;
    stLENS2_428[283].fEnergy := 14573.391729; stLENS2_428[283].fLow := 16.630188; stLENS2_428[283].fHigh := 59.651874;
    stLENS2_428[284].fEnergy := 14602.567679; stLENS2_428[284].fLow := 16.568145; stLENS2_428[284].fHigh := 59.270489;
    stLENS2_428[285].fEnergy := 14631.802039; stLENS2_428[285].fLow := 16.506334; stLENS2_428[285].fHigh := 58.891541;
    stLENS2_428[286].fEnergy := 14661.094926; stLENS2_428[286].fLow := 16.444754; stLENS2_428[286].fHigh := 58.515017;
    stLENS2_428[287].fEnergy := 14690.446458; stLENS2_428[287].fLow := 16.383403; stLENS2_428[287].fHigh := 58.140899;
    stLENS2_428[288].fEnergy := 14719.856751; stLENS2_428[288].fLow := 16.322281; stLENS2_428[288].fHigh := 57.769174;
    stLENS2_428[289].fEnergy := 14749.325924; stLENS2_428[289].fLow := 16.261387; stLENS2_428[289].fHigh := 57.399826;
    stLENS2_428[290].fEnergy := 14778.854094; stLENS2_428[290].fLow := 16.200721; stLENS2_428[290].fHigh := 57.032838;
    stLENS2_428[291].fEnergy := 14808.441380; stLENS2_428[291].fLow := 16.140280; stLENS2_428[291].fHigh := 56.668198;
    stLENS2_428[292].fEnergy := 14838.087899; stLENS2_428[292].fLow := 16.080066; stLENS2_428[292].fHigh := 56.184807;
    stLENS2_428[293].fEnergy := 14867.793771; stLENS2_428[293].fLow := 16.020075; stLENS2_428[293].fHigh := 55.890485;
    stLENS2_428[294].fEnergy := 14897.559114; stLENS2_428[294].fLow := 15.960309; stLENS2_428[294].fHigh := 55.597866;
    stLENS2_428[295].fEnergy := 14927.384047; stLENS2_428[295].fLow := 15.900766; stLENS2_428[295].fHigh := 55.306939;
    stLENS2_428[296].fEnergy := 14957.268690; stLENS2_428[296].fLow := 15.841444; stLENS2_428[296].fHigh := 55.017695;
    stLENS2_428[297].fEnergy := 14987.213162; stLENS2_428[297].fLow := 15.782345; stLENS2_428[297].fHigh := 54.730122;
    stLENS2_428[298].fEnergy := 15017.217582; stLENS2_428[298].fLow := 15.723465; stLENS2_428[298].fHigh := 54.444210;
    stLENS2_428[299].fEnergy := 15047.282072; stLENS2_428[299].fLow := 15.664805; stLENS2_428[299].fHigh := 54.159948;
    stLENS2_428[300].fEnergy := 15077.406751; stLENS2_428[300].fLow := 15.606364; stLENS2_428[300].fHigh := 53.877327;
    stLENS2_428[301].fEnergy := 15107.591739; stLENS2_428[301].fLow := 15.548141; stLENS2_428[301].fHigh := 53.596337;
    stLENS2_428[302].fEnergy := 15137.837158; stLENS2_428[302].fLow := 15.490136; stLENS2_428[302].fHigh := 53.316967;
    stLENS2_428[303].fEnergy := 15168.143128; stLENS2_428[303].fLow := 15.432346; stLENS2_428[303].fHigh := 53.039206;
    stLENS2_428[304].fEnergy := 15198.509771; stLENS2_428[304].fLow := 15.374773; stLENS2_428[304].fHigh := 52.763046;
    stLENS2_428[305].fEnergy := 15228.937208; stLENS2_428[305].fLow := 15.317414; stLENS2_428[305].fHigh := 52.488476;
    stLENS2_428[306].fEnergy := 15259.425560; stLENS2_428[306].fLow := 15.260269; stLENS2_428[306].fHigh := 52.215486;
    stLENS2_428[307].fEnergy := 15289.974951; stLENS2_428[307].fLow := 15.203337; stLENS2_428[307].fHigh := 51.944067;
    stLENS2_428[308].fEnergy := 15320.585501; stLENS2_428[308].fLow := 15.146618; stLENS2_428[308].fHigh := 51.674209;
    stLENS2_428[309].fEnergy := 15351.257334; stLENS2_428[309].fLow := 15.090110; stLENS2_428[309].fHigh := 51.405902;
    stLENS2_428[310].fEnergy := 15381.990571; stLENS2_428[310].fLow := 15.033813; stLENS2_428[310].fHigh := 51.139136;
    stLENS2_428[311].fEnergy := 15412.785337; stLENS2_428[311].fLow := 14.977726; stLENS2_428[311].fHigh := 50.873902;
    stLENS2_428[312].fEnergy := 15443.641754; stLENS2_428[312].fLow := 14.921849; stLENS2_428[312].fHigh := 50.610190;
    stLENS2_428[313].fEnergy := 15474.559945; stLENS2_428[313].fLow := 14.866179; stLENS2_428[313].fHigh := 50.347992;
    stLENS2_428[314].fEnergy := 15505.540035; stLENS2_428[314].fLow := 14.810718; stLENS2_428[314].fHigh := 50.087297;
    stLENS2_428[315].fEnergy := 15536.582147; stLENS2_428[315].fLow := 14.755463; stLENS2_428[315].fHigh := 49.828097;
    stLENS2_428[316].fEnergy := 15567.686405; stLENS2_428[316].fLow := 14.700415; stLENS2_428[316].fHigh := 49.570382;
    stLENS2_428[317].fEnergy := 15598.852934; stLENS2_428[317].fLow := 14.645572; stLENS2_428[317].fHigh := 49.314143;
    stLENS2_428[318].fEnergy := 15630.081858; stLENS2_428[318].fLow := 14.590933; stLENS2_428[318].fHigh := 49.059371;
    stLENS2_428[319].fEnergy := 15661.373303; stLENS2_428[319].fLow := 14.536499; stLENS2_428[319].fHigh := 48.806056;
    stLENS2_428[320].fEnergy := 15692.727393; stLENS2_428[320].fLow := 14.482267; stLENS2_428[320].fHigh := 48.554191;
    stLENS2_428[321].fEnergy := 15724.144254; stLENS2_428[321].fLow := 14.428238; stLENS2_428[321].fHigh := 48.303765;
    stLENS2_428[322].fEnergy := 15755.624012; stLENS2_428[322].fLow := 14.374410; stLENS2_428[322].fHigh := 48.054770;
    stLENS2_428[323].fEnergy := 15787.166792; stLENS2_428[323].fLow := 14.320783; stLENS2_428[323].fHigh := 47.807198;
    stLENS2_428[324].fEnergy := 15818.772721; stLENS2_428[324].fLow := 14.267357; stLENS2_428[324].fHigh := 47.561039;
    stLENS2_428[325].fEnergy := 15850.441925; stLENS2_428[325].fLow := 14.214129; stLENS2_428[325].fHigh := 47.316285;
    stLENS2_428[326].fEnergy := 15882.174531; stLENS2_428[326].fLow := 14.161100; stLENS2_428[326].fHigh := 47.072926;
    stLENS2_428[327].fEnergy := 15913.970666; stLENS2_428[327].fLow := 14.108269; stLENS2_428[327].fHigh := 46.830956;
    stLENS2_428[328].fEnergy := 15945.830456; stLENS2_428[328].fLow := 14.055635; stLENS2_428[328].fHigh := 46.590364;
    stLENS2_428[329].fEnergy := 15977.754030; stLENS2_428[329].fLow := 14.003198; stLENS2_428[329].fHigh := 46.351143;
    stLENS2_428[330].fEnergy := 16009.741515; stLENS2_428[330].fLow := 13.950956; stLENS2_428[330].fHigh := 46.113284;
    stLENS2_428[331].fEnergy := 16041.793039; stLENS2_428[331].fLow := 13.898909; stLENS2_428[331].fHigh := 45.876779;
    stLENS2_428[332].fEnergy := 16073.908730; stLENS2_428[332].fLow := 13.847056; stLENS2_428[332].fHigh := 45.641619;
    stLENS2_428[333].fEnergy := 16106.088717; stLENS2_428[333].fLow := 13.795396; stLENS2_428[333].fHigh := 45.407796;
    stLENS2_428[334].fEnergy := 16138.333128; stLENS2_428[334].fLow := 13.743930; stLENS2_428[334].fHigh := 45.175302;
    stLENS2_428[335].fEnergy := 16170.642092; stLENS2_428[335].fLow := 13.692655; stLENS2_428[335].fHigh := 44.944129;
    stLENS2_428[336].fEnergy := 16203.015739; stLENS2_428[336].fLow := 13.641571; stLENS2_428[336].fHigh := 44.714268;
    stLENS2_428[337].fEnergy := 16235.454198; stLENS2_428[337].fLow := 13.590679; stLENS2_428[337].fHigh := 44.485713;
    stLENS2_428[338].fEnergy := 16267.957599; stLENS2_428[338].fLow := 13.539976; stLENS2_428[338].fHigh := 44.258454;
    stLENS2_428[339].fEnergy := 16300.526072; stLENS2_428[339].fLow := 13.489462; stLENS2_428[339].fHigh := 44.032483;
    stLENS2_428[340].fEnergy := 16333.159747; stLENS2_428[340].fLow := 13.439137; stLENS2_428[340].fHigh := 43.807794;
    stLENS2_428[341].fEnergy := 16365.858755; stLENS2_428[341].fLow := 13.388999; stLENS2_428[341].fHigh := 43.584377;
    stLENS2_428[342].fEnergy := 16398.623226; stLENS2_428[342].fLow := 13.339048; stLENS2_428[342].fHigh := 43.362226;
    stLENS2_428[343].fEnergy := 16431.453291; stLENS2_428[343].fLow := 13.289284; stLENS2_428[343].fHigh := 43.141332;
    stLENS2_428[344].fEnergy := 16464.349083; stLENS2_428[344].fLow := 13.239706; stLENS2_428[344].fHigh := 42.921688;
    stLENS2_428[345].fEnergy := 16497.310732; stLENS2_428[345].fLow := 13.190312; stLENS2_428[345].fHigh := 42.703286;
    stLENS2_428[346].fEnergy := 16530.338370; stLENS2_428[346].fLow := 13.141103; stLENS2_428[346].fHigh := 42.486119;
    stLENS2_428[347].fEnergy := 16563.432129; stLENS2_428[347].fLow := 13.092077; stLENS2_428[347].fHigh := 42.270178;
    stLENS2_428[348].fEnergy := 16596.592142; stLENS2_428[348].fLow := 13.043234; stLENS2_428[348].fHigh := 42.055457;
    stLENS2_428[349].fEnergy := 16629.818542; stLENS2_428[349].fLow := 12.994574; stLENS2_428[349].fHigh := 41.841949;
    stLENS2_428[350].fEnergy := 16663.111461; stLENS2_428[350].fLow := 12.946094; stLENS2_428[350].fHigh := 41.629645;
    stLENS2_428[351].fEnergy := 16696.471032; stLENS2_428[351].fLow := 12.897796; stLENS2_428[351].fHigh := 41.418538;
    stLENS2_428[352].fEnergy := 16729.897390; stLENS2_428[352].fLow := 12.849678; stLENS2_428[352].fHigh := 41.208622;
    stLENS2_428[353].fEnergy := 16763.390666; stLENS2_428[353].fLow := 12.801740; stLENS2_428[353].fHigh := 40.999888;
    stLENS2_428[354].fEnergy := 16796.950997; stLENS2_428[354].fLow := 12.753980; stLENS2_428[354].fHigh := 40.792330;
    stLENS2_428[355].fEnergy := 16830.578515; stLENS2_428[355].fLow := 12.706399; stLENS2_428[355].fHigh := 40.585941;
    stLENS2_428[356].fEnergy := 16864.273356; stLENS2_428[356].fLow := 12.658995; stLENS2_428[356].fHigh := 40.380713;
    stLENS2_428[357].fEnergy := 16898.035654; stLENS2_428[357].fLow := 12.611767; stLENS2_428[357].fHigh := 40.176639;
    stLENS2_428[358].fEnergy := 16931.865544; stLENS2_428[358].fLow := 12.564717; stLENS2_428[358].fHigh := 39.973712;
    stLENS2_428[359].fEnergy := 16965.763161; stLENS2_428[359].fLow := 12.517841; stLENS2_428[359].fHigh := 39.771926;
    stLENS2_428[360].fEnergy := 16999.728641; stLENS2_428[360].fLow := 12.471141; stLENS2_428[360].fHigh := 39.571274;
    stLENS2_428[361].fEnergy := 17033.762121; stLENS2_428[361].fLow := 12.424614; stLENS2_428[361].fHigh := 39.371747;
    stLENS2_428[362].fEnergy := 17067.863735; stLENS2_428[362].fLow := 12.378262; stLENS2_428[362].fHigh := 39.173341;
    stLENS2_428[363].fEnergy := 17102.033621; stLENS2_428[363].fLow := 12.332082; stLENS2_428[363].fHigh := 38.976047;
    stLENS2_428[364].fEnergy := 17136.271915; stLENS2_428[364].fLow := 12.286074; stLENS2_428[364].fHigh := 38.779860;
    stLENS2_428[365].fEnergy := 17170.578755; stLENS2_428[365].fLow := 12.240239; stLENS2_428[365].fHigh := 38.584772;
    stLENS2_428[366].fEnergy := 17204.954276; stLENS2_428[366].fLow := 12.194574; stLENS2_428[366].fHigh := 38.390777;
    stLENS2_428[367].fEnergy := 17239.398618; stLENS2_428[367].fLow := 12.149079; stLENS2_428[367].fHigh := 38.197868;
    stLENS2_428[368].fEnergy := 17273.911917; stLENS2_428[368].fLow := 12.103754; stLENS2_428[368].fHigh := 38.006039;
    stLENS2_428[369].fEnergy := 17308.494311; stLENS2_428[369].fLow := 12.058599; stLENS2_428[369].fHigh := 37.815282;
    stLENS2_428[370].fEnergy := 17343.145940; stLENS2_428[370].fLow := 12.013612; stLENS2_428[370].fHigh := 37.625593;
    stLENS2_428[371].fEnergy := 17377.866941; stLENS2_428[371].fLow := 11.968792; stLENS2_428[371].fHigh := 37.436963;
    stLENS2_428[372].fEnergy := 17412.657454; stLENS2_428[372].fLow := 11.924140; stLENS2_428[372].fHigh := 37.249387;
    stLENS2_428[373].fEnergy := 17447.517618; stLENS2_428[373].fLow := 11.879654; stLENS2_428[373].fHigh := 37.062859;
    stLENS2_428[374].fEnergy := 17482.447571; stLENS2_428[374].fLow := 11.835335; stLENS2_428[374].fHigh := 36.877371;
    stLENS2_428[375].fEnergy := 17517.447455; stLENS2_428[375].fLow := 11.791180; stLENS2_428[375].fHigh := 36.692918;
    stLENS2_428[376].fEnergy := 17552.517408; stLENS2_428[376].fLow := 11.747191; stLENS2_428[376].fHigh := 36.509494;
    stLENS2_428[377].fEnergy := 17587.657571; stLENS2_428[377].fLow := 11.703365; stLENS2_428[377].fHigh := 36.327092;
    stLENS2_428[378].fEnergy := 17622.868085; stLENS2_428[378].fLow := 11.659704; stLENS2_428[378].fHigh := 36.145707;
    stLENS2_428[379].fEnergy := 17658.149090; stLENS2_428[379].fLow := 11.616205; stLENS2_428[379].fHigh := 35.965331;
    stLENS2_428[380].fEnergy := 17693.500728; stLENS2_428[380].fLow := 11.572868; stLENS2_428[380].fHigh := 35.785959;
    stLENS2_428[381].fEnergy := 17728.923140; stLENS2_428[381].fLow := 11.529693; stLENS2_428[381].fHigh := 35.607585;
    stLENS2_428[382].fEnergy := 17764.416468; stLENS2_428[382].fLow := 11.486679; stLENS2_428[382].fHigh := 35.430203;
    stLENS2_428[383].fEnergy := 17799.980854; stLENS2_428[383].fLow := 11.443825; stLENS2_428[383].fHigh := 35.253807;
    stLENS2_428[384].fEnergy := 17835.616439; stLENS2_428[384].fLow := 11.401131; stLENS2_428[384].fHigh := 35.078391;
    stLENS2_428[385].fEnergy := 17871.323367; stLENS2_428[385].fLow := 11.358597; stLENS2_428[385].fHigh := 34.903949;
    stLENS2_428[386].fEnergy := 17907.101780; stLENS2_428[386].fLow := 11.316221; stLENS2_428[386].fHigh := 34.730476;
    stLENS2_428[387].fEnergy := 17942.951822; stLENS2_428[387].fLow := 11.274004; stLENS2_428[387].fHigh := 34.557964;
    stLENS2_428[388].fEnergy := 17978.873635; stLENS2_428[388].fLow := 11.231944; stLENS2_428[388].fHigh := 34.386410;
    stLENS2_428[389].fEnergy := 18014.867364; stLENS2_428[389].fLow := 11.190040; stLENS2_428[389].fHigh := 34.215806;
    stLENS2_428[390].fEnergy := 18050.933153; stLENS2_428[390].fLow := 11.148294; stLENS2_428[390].fHigh := 34.046148;
    stLENS2_428[391].fEnergy := 18087.071145; stLENS2_428[391].fLow := 11.106702; stLENS2_428[391].fHigh := 33.877429;
    stLENS2_428[392].fEnergy := 18123.281486; stLENS2_428[392].fLow := 11.065266; stLENS2_428[392].fHigh := 33.709643;
    stLENS2_428[393].fEnergy := 18159.564319; stLENS2_428[393].fLow := 11.023985; stLENS2_428[393].fHigh := 33.542787;
    stLENS2_428[394].fEnergy := 18195.919791; stLENS2_428[394].fLow := 10.982858; stLENS2_428[394].fHigh := 33.376853;
    stLENS2_428[395].fEnergy := 18232.348047; stLENS2_428[395].fLow := 10.941884; stLENS2_428[395].fHigh := 33.211836;
    stLENS2_428[396].fEnergy := 18268.849232; stLENS2_428[396].fLow := 10.901063; stLENS2_428[396].fHigh := 33.047731;
    stLENS2_428[397].fEnergy := 18305.423493; stLENS2_428[397].fLow := 10.860394; stLENS2_428[397].fHigh := 32.884532;
    stLENS2_428[398].fEnergy := 18342.070975; stLENS2_428[398].fLow := 10.819877; stLENS2_428[398].fHigh := 32.722234;
    stLENS2_428[399].fEnergy := 18378.791826; stLENS2_428[399].fLow := 10.779511; stLENS2_428[399].fHigh := 32.560831;
    stLENS2_428[400].fEnergy := 18415.586191; stLENS2_428[400].fLow := 10.739296; stLENS2_428[400].fHigh := 32.400319;
    stLENS2_428[401].fEnergy := 18452.454219; stLENS2_428[401].fLow := 10.699230; stLENS2_428[401].fHigh := 32.240691;
    stLENS2_428[402].fEnergy := 18489.396057; stLENS2_428[402].fLow := 10.659315; stLENS2_428[402].fHigh := 32.081943;
    stLENS2_428[403].fEnergy := 18526.411853; stLENS2_428[403].fLow := 10.619548; stLENS2_428[403].fHigh := 31.924070;
    stLENS2_428[404].fEnergy := 18563.501754; stLENS2_428[404].fLow := 10.579929; stLENS2_428[404].fHigh := 31.767065;
    stLENS2_428[405].fEnergy := 18600.665909; stLENS2_428[405].fLow := 10.540459; stLENS2_428[405].fHigh := 31.610924;
    stLENS2_428[406].fEnergy := 18637.904467; stLENS2_428[406].fLow := 10.501135; stLENS2_428[406].fHigh := 31.455642;
    stLENS2_428[407].fEnergy := 18675.217577; stLENS2_428[407].fLow := 10.461958; stLENS2_428[407].fHigh := 31.301213;
    stLENS2_428[408].fEnergy := 18712.605388; stLENS2_428[408].fLow := 10.422928; stLENS2_428[408].fHigh := 31.147633;
    stLENS2_428[409].fEnergy := 18750.068048; stLENS2_428[409].fLow := 10.384043; stLENS2_428[409].fHigh := 30.994897;
    stLENS2_428[410].fEnergy := 18787.605710; stLENS2_428[410].fLow := 10.345303; stLENS2_428[410].fHigh := 30.842998;
    stLENS2_428[411].fEnergy := 18825.218521; stLENS2_428[411].fLow := 10.306707; stLENS2_428[411].fHigh := 30.691934;
    stLENS2_428[412].fEnergy := 18862.906634; stLENS2_428[412].fLow := 10.268256; stLENS2_428[412].fHigh := 30.541698;
    stLENS2_428[413].fEnergy := 18900.670198; stLENS2_428[413].fLow := 10.229948; stLENS2_428[413].fHigh := 30.392285;
    stLENS2_428[414].fEnergy := 18938.509365; stLENS2_428[414].fLow := 10.191783; stLENS2_428[414].fHigh := 30.243691;
    stLENS2_428[415].fEnergy := 18976.424286; stLENS2_428[415].fLow := 10.153760; stLENS2_428[415].fHigh := 30.095911;
    stLENS2_428[416].fEnergy := 19014.415113; stLENS2_428[416].fLow := 10.115880; stLENS2_428[416].fHigh := 29.948940;
    stLENS2_428[417].fEnergy := 19052.481997; stLENS2_428[417].fLow := 10.078140; stLENS2_428[417].fHigh := 29.802773;
    stLENS2_428[418].fEnergy := 19090.625092; stLENS2_428[418].fLow := 10.040541; stLENS2_428[418].fHigh := 29.657405;
    stLENS2_428[419].fEnergy := 19128.844549; stLENS2_428[419].fLow := 10.003083; stLENS2_428[419].fHigh := 29.512833;
    stLENS2_428[420].fEnergy := 19167.140521; stLENS2_428[420].fLow := 9.965764; stLENS2_428[420].fHigh := 29.369050;
    stLENS2_428[421].fEnergy := 19205.513162; stLENS2_428[421].fLow := 9.928585; stLENS2_428[421].fHigh := 29.226052;
    stLENS2_428[422].fEnergy := 19243.962625; stLENS2_428[422].fLow := 9.891544; stLENS2_428[422].fHigh := 29.083835;
    stLENS2_428[423].fEnergy := 19282.489064; stLENS2_428[423].fLow := 9.854642; stLENS2_428[423].fHigh := 28.942394;
    stLENS2_428[424].fEnergy := 19321.092632; stLENS2_428[424].fLow := 9.817877; stLENS2_428[424].fHigh := 28.801725;
    stLENS2_428[425].fEnergy := 19359.773486; stLENS2_428[425].fLow := 9.781249; stLENS2_428[425].fHigh := 28.661822;
    stLENS2_428[426].fEnergy := 19398.531778; stLENS2_428[426].fLow := 9.744758; stLENS2_428[426].fHigh := 28.522682;
    stLENS2_428[427].fEnergy := 19437.367665; stLENS2_428[427].fLow := 9.708403; stLENS2_428[427].fHigh := 28.384299;
    stLENS2_428[428].fEnergy := 19476.281301; stLENS2_428[428].fLow := 9.672184; stLENS2_428[428].fHigh := 28.246670;
    stLENS2_428[429].fEnergy := 19515.272842; stLENS2_428[429].fLow := 9.636100; stLENS2_428[429].fHigh := 28.109790;
    stLENS2_428[430].fEnergy := 19554.342444; stLENS2_428[430].fLow := 9.600150; stLENS2_428[430].fHigh := 27.973654;
    stLENS2_428[431].fEnergy := 19593.490264; stLENS2_428[431].fLow := 9.564335; stLENS2_428[431].fHigh := 27.838258;
    stLENS2_428[432].fEnergy := 19632.716457; stLENS2_428[432].fLow := 9.528653; stLENS2_428[432].fHigh := 27.703598;
    stLENS2_428[433].fEnergy := 19672.021182; stLENS2_428[433].fLow := 9.493104; stLENS2_428[433].fHigh := 27.569669;
    stLENS2_428[434].fEnergy := 19711.404594; stLENS2_428[434].fLow := 9.457688; stLENS2_428[434].fHigh := 27.436467;
    stLENS2_428[435].fEnergy := 19750.866853; stLENS2_428[435].fLow := 9.422404; stLENS2_428[435].fHigh := 27.303989;
    stLENS2_428[436].fEnergy := 19790.408115; stLENS2_428[436].fLow := 9.387252; stLENS2_428[436].fHigh := 27.172228;
    stLENS2_428[437].fEnergy := 19830.028538; stLENS2_428[437].fLow := 9.352231; stLENS2_428[437].fHigh := 27.041182;
    stLENS2_428[438].fEnergy := 19869.728282; stLENS2_428[438].fLow := 9.317340; stLENS2_428[438].fHigh := 26.910846;
    stLENS2_428[439].fEnergy := 19909.507504; stLENS2_428[439].fLow := 9.282580; stLENS2_428[439].fHigh := 26.781216;
    stLENS2_428[440].fEnergy := 19949.366365; stLENS2_428[440].fLow := 9.247949; stLENS2_428[440].fHigh := 26.652288;
    stLENS2_428[441].fEnergy := 19989.305023; stLENS2_428[441].fLow := 9.213448; stLENS2_428[441].fHigh := 26.524057;
    stLENS2_428[442].fEnergy := 20029.323638; stLENS2_428[442].fLow := 9.179075; stLENS2_428[442].fHigh := 26.396520;
    stLENS2_428[443].fEnergy := 20069.422371; stLENS2_428[443].fLow := 9.144830; stLENS2_428[443].fHigh := 26.269672;
    stLENS2_428[444].fEnergy := 20109.601381; stLENS2_428[444].fLow := 9.110713; stLENS2_428[444].fHigh := 26.143510;
    stLENS2_428[445].fEnergy := 20149.860830; stLENS2_428[445].fLow := 9.076724; stLENS2_428[445].fHigh := 26.018029;
    stLENS2_428[446].fEnergy := 20190.200878; stLENS2_428[446].fLow := 9.042861; stLENS2_428[446].fHigh := 25.893225;
    stLENS2_428[447].fEnergy := 20230.621687; stLENS2_428[447].fLow := 9.009125; stLENS2_428[447].fHigh := 25.769095;
    stLENS2_428[448].fEnergy := 20271.123419; stLENS2_428[448].fLow := 8.975514; stLENS2_428[448].fHigh := 25.645634;
    stLENS2_428[449].fEnergy := 20311.706235; stLENS2_428[449].fLow := 8.942029; stLENS2_428[449].fHigh := 25.522839;
    stLENS2_428[450].fEnergy := 20352.370298; stLENS2_428[450].fLow := 8.908669; stLENS2_428[450].fHigh := 25.400706;
    stLENS2_428[451].fEnergy := 20393.115770; stLENS2_428[451].fLow := 8.875433; stLENS2_428[451].fHigh := 25.279230;
    stLENS2_428[452].fEnergy := 20433.942815; stLENS2_428[452].fLow := 8.842322; stLENS2_428[452].fHigh := 25.158408;
    stLENS2_428[453].fEnergy := 20474.851596; stLENS2_428[453].fLow := 8.809334; stLENS2_428[453].fHigh := 25.038237;
    stLENS2_428[454].fEnergy := 20515.842276; stLENS2_428[454].fLow := 8.776468; stLENS2_428[454].fHigh := 24.918711;
    stLENS2_428[455].fEnergy := 20556.915020; stLENS2_428[455].fLow := 8.743726; stLENS2_428[455].fHigh := 24.799829;
    stLENS2_428[456].fEnergy := 20598.069991; stLENS2_428[456].fLow := 8.711106; stLENS2_428[456].fHigh := 24.681585;
    stLENS2_428[457].fEnergy := 20639.307355; stLENS2_428[457].fLow := 8.678607; stLENS2_428[457].fHigh := 24.563976;
    stLENS2_428[458].fEnergy := 20680.627276; stLENS2_428[458].fLow := 8.646229; stLENS2_428[458].fHigh := 24.446998;
    stLENS2_428[459].fEnergy := 20722.029919; stLENS2_428[459].fLow := 8.613973; stLENS2_428[459].fHigh := 24.330648;
    stLENS2_428[460].fEnergy := 20763.515451; stLENS2_428[460].fLow := 8.581837; stLENS2_428[460].fHigh := 24.214922;
    stLENS2_428[461].fEnergy := 20805.084036; stLENS2_428[461].fLow := 8.549820; stLENS2_428[461].fHigh := 24.099816;
    stLENS2_428[462].fEnergy := 20846.735842; stLENS2_428[462].fLow := 8.517923; stLENS2_428[462].fHigh := 23.985327;
    stLENS2_428[463].fEnergy := 20888.471035; stLENS2_428[463].fLow := 8.486145; stLENS2_428[463].fHigh := 23.871452;
    stLENS2_428[464].fEnergy := 20930.289782; stLENS2_428[464].fLow := 8.454486; stLENS2_428[464].fHigh := 23.758186;
    stLENS2_428[465].fEnergy := 20972.192250; stLENS2_428[465].fLow := 8.422945; stLENS2_428[465].fHigh := 23.645525;
    stLENS2_428[466].fEnergy := 21014.178607; stLENS2_428[466].fLow := 8.391521; stLENS2_428[466].fHigh := 23.533468;
    stLENS2_428[467].fEnergy := 21056.249021; stLENS2_428[467].fLow := 8.360215; stLENS2_428[467].fHigh := 23.422009;
    stLENS2_428[468].fEnergy := 21098.403659; stLENS2_428[468].fLow := 8.329025; stLENS2_428[468].fHigh := 23.311146;
    stLENS2_428[469].fEnergy := 21140.642692; stLENS2_428[469].fLow := 8.297952; stLENS2_428[469].fHigh := 23.200875;
    stLENS2_428[470].fEnergy := 21182.966286; stLENS2_428[470].fLow := 8.266994; stLENS2_428[470].fHigh := 23.091193;
    stLENS2_428[471].fEnergy := 21225.374613; stLENS2_428[471].fLow := 8.236153; stLENS2_428[471].fHigh := 22.982095;
    stLENS2_428[472].fEnergy := 21267.867841; stLENS2_428[472].fLow := 8.205426; stLENS2_428[472].fHigh := 22.873580;
    stLENS2_428[473].fEnergy := 21310.446141; stLENS2_428[473].fLow := 8.174814; stLENS2_428[473].fHigh := 22.765643;
    stLENS2_428[474].fEnergy := 21353.109683; stLENS2_428[474].fLow := 8.144316; stLENS2_428[474].fHigh := 22.658281;
    stLENS2_428[475].fEnergy := 21395.858637; stLENS2_428[475].fLow := 8.113932; stLENS2_428[475].fHigh := 22.551491;
    stLENS2_428[476].fEnergy := 21438.693174; stLENS2_428[476].fLow := 8.083661; stLENS2_428[476].fHigh := 22.445269;
    stLENS2_428[477].fEnergy := 21481.613467; stLENS2_428[477].fLow := 8.053503; stLENS2_428[477].fHigh := 22.339612;
    stLENS2_428[478].fEnergy := 21524.619686; stLENS2_428[478].fLow := 8.023458; stLENS2_428[478].fHigh := 22.234517;
    stLENS2_428[479].fEnergy := 21567.712003; stLENS2_428[479].fLow := 7.993524; stLENS2_428[479].fHigh := 22.129981;
    stLENS2_428[480].fEnergy := 21610.890591; stLENS2_428[480].fLow := 7.963703; stLENS2_428[480].fHigh := 22.026001;
    stLENS2_428[481].fEnergy := 21654.155623; stLENS2_428[481].fLow := 7.933993; stLENS2_428[481].fHigh := 21.922572;
    stLENS2_428[482].fEnergy := 21697.507271; stLENS2_428[482].fLow := 7.904393; stLENS2_428[482].fHigh := 21.819692;
    stLENS2_428[483].fEnergy := 21740.945710; stLENS2_428[483].fLow := 7.874904; stLENS2_428[483].fHigh := 21.717358;
    stLENS2_428[484].fEnergy := 21784.471112; stLENS2_428[484].fLow := 7.845525; stLENS2_428[484].fHigh := 21.615567;
    stLENS2_428[485].fEnergy := 21828.083652; stLENS2_428[485].fLow := 7.816256; stLENS2_428[485].fHigh := 21.514316;
    stLENS2_428[486].fEnergy := 21871.783505; stLENS2_428[486].fLow := 7.787095; stLENS2_428[486].fHigh := 21.413600;
    stLENS2_428[487].fEnergy := 21915.570845; stLENS2_428[487].fLow := 7.758044; stLENS2_428[487].fHigh := 21.313418;
    stLENS2_428[488].fEnergy := 21959.445847; stLENS2_428[488].fLow := 7.729101; stLENS2_428[488].fHigh := 21.213767;
    stLENS2_428[489].fEnergy := 22003.408687; stLENS2_428[489].fLow := 7.700266; stLENS2_428[489].fHigh := 21.114642;
    stLENS2_428[490].fEnergy := 22047.459540; stLENS2_428[490].fLow := 7.671538; stLENS2_428[490].fHigh := 21.016042;
    stLENS2_428[491].fEnergy := 22091.598584; stLENS2_428[491].fLow := 7.642918; stLENS2_428[491].fHigh := 20.917963;
    stLENS2_428[492].fEnergy := 22135.825994; stLENS2_428[492].fLow := 7.614404; stLENS2_428[492].fHigh := 20.820402;
    stLENS2_428[493].fEnergy := 22180.141947; stLENS2_428[493].fLow := 7.585997; stLENS2_428[493].fHigh := 20.723356;
    stLENS2_428[494].fEnergy := 22224.546620; stLENS2_428[494].fLow := 7.557696; stLENS2_428[494].fHigh := 20.626822;
    stLENS2_428[495].fEnergy := 22269.040192; stLENS2_428[495].fLow := 7.529500; stLENS2_428[495].fHigh := 20.530797;
    stLENS2_428[496].fEnergy := 22313.622841; stLENS2_428[496].fLow := 7.501410; stLENS2_428[496].fHigh := 20.435279;
    stLENS2_428[497].fEnergy := 22358.294743; stLENS2_428[497].fLow := 7.473424; stLENS2_428[497].fHigh := 20.340264;
    stLENS2_428[498].fEnergy := 22403.056079; stLENS2_428[498].fLow := 7.445543; stLENS2_428[498].fHigh := 20.245750;
    stLENS2_428[499].fEnergy := 22447.907027; stLENS2_428[499].fLow := 7.417766; stLENS2_428[499].fHigh := 20.151733;
    stLENS2_428[500].fEnergy := 22492.847767; stLENS2_428[500].fLow := 7.390092; stLENS2_428[500].fHigh := 20.058211;
    stLENS2_428[501].fEnergy := 22537.878478; stLENS2_428[501].fLow := 7.362522; stLENS2_428[501].fHigh := 19.965181;
    stLENS2_428[502].fEnergy := 22582.999341; stLENS2_428[502].fLow := 7.335054; stLENS2_428[502].fHigh := 19.872641;
    stLENS2_428[503].fEnergy := 22628.210536; stLENS2_428[503].fLow := 7.307689; stLENS2_428[503].fHigh := 19.780586;
    stLENS2_428[504].fEnergy := 22673.512244; stLENS2_428[504].fLow := 7.280427; stLENS2_428[504].fHigh := 19.689015;
    stLENS2_428[505].fEnergy := 22718.904645; stLENS2_428[505].fLow := 7.253265; stLENS2_428[505].fHigh := 19.597925;
    stLENS2_428[506].fEnergy := 22764.387923; stLENS2_428[506].fLow := 7.226205; stLENS2_428[506].fHigh := 19.507313;
    stLENS2_428[507].fEnergy := 22809.962258; stLENS2_428[507].fLow := 7.199247; stLENS2_428[507].fHigh := 19.417176;
    stLENS2_428[508].fEnergy := 22855.627833; stLENS2_428[508].fLow := 7.172388; stLENS2_428[508].fHigh := 19.327512;
    stLENS2_428[509].fEnergy := 22901.384830; stLENS2_428[509].fLow := 7.145630; stLENS2_428[509].fHigh := 19.238317;
    stLENS2_428[510].fEnergy := 22947.233433; stLENS2_428[510].fLow := 7.118972; stLENS2_428[510].fHigh := 19.149590;
    stLENS2_428[511].fEnergy := 22993.173825; stLENS2_428[511].fLow := 7.092413; stLENS2_428[511].fHigh := 19.061327;
    stLENS2_428[512].fEnergy := 23039.206190; stLENS2_428[512].fLow := 7.065953; stLENS2_428[512].fHigh := 18.973526;
    stLENS2_428[513].fEnergy := 23085.330711; stLENS2_428[513].fLow := 7.039592; stLENS2_428[513].fHigh := 18.886184;
    stLENS2_428[514].fEnergy := 23131.547574; stLENS2_428[514].fLow := 7.013329; stLENS2_428[514].fHigh := 18.799299;
    stLENS2_428[515].fEnergy := 23177.856963; stLENS2_428[515].fLow := 6.987165; stLENS2_428[515].fHigh := 18.712868;
    stLENS2_428[516].fEnergy := 23224.259064; stLENS2_428[516].fLow := 6.961097; stLENS2_428[516].fHigh := 18.626889;
    stLENS2_428[517].fEnergy := 23270.754061; stLENS2_428[517].fLow := 6.935128; stLENS2_428[517].fHigh := 18.541358;
    stLENS2_428[518].fEnergy := 23317.342142; stLENS2_428[518].fLow := 6.909255; stLENS2_428[518].fHigh := 18.456273;
    stLENS2_428[519].fEnergy := 23364.023492; stLENS2_428[519].fLow := 6.883478; stLENS2_428[519].fHigh := 18.371633;
    stLENS2_428[520].fEnergy := 23410.798298; stLENS2_428[520].fLow := 6.857798; stLENS2_428[520].fHigh := 18.287433;
    stLENS2_428[521].fEnergy := 23457.666748; stLENS2_428[521].fLow := 6.832213; stLENS2_428[521].fHigh := 18.203672;
    stLENS2_428[522].fEnergy := 23504.629028; stLENS2_428[522].fLow := 6.806724; stLENS2_428[522].fHigh := 18.120347;
    stLENS2_428[523].fEnergy := 23551.685327; stLENS2_428[523].fLow := 6.781330; stLENS2_428[523].fHigh := 18.037457;
    stLENS2_428[524].fEnergy := 23598.835832; stLENS2_428[524].fLow := 6.756031; stLENS2_428[524].fHigh := 17.954997;
    stLENS2_428[525].fEnergy := 23646.080733; stLENS2_428[525].fLow := 6.730826; stLENS2_428[525].fHigh := 17.872966;
    stLENS2_428[526].fEnergy := 23693.420218; stLENS2_428[526].fLow := 6.705715; stLENS2_428[526].fHigh := 17.791362;
    stLENS2_428[527].fEnergy := 23740.854477; stLENS2_428[527].fLow := 6.680698; stLENS2_428[527].fHigh := 17.710181;
    stLENS2_428[528].fEnergy := 23788.383699; stLENS2_428[528].fLow := 6.655775; stLENS2_428[528].fHigh := 17.629422;
    stLENS2_428[529].fEnergy := 23836.008075; stLENS2_428[529].fLow := 6.630944; stLENS2_428[529].fHigh := 17.549083;
    stLENS2_428[530].fEnergy := 23883.727795; stLENS2_428[530].fLow := 6.606206; stLENS2_428[530].fHigh := 17.469160;
    stLENS2_428[531].fEnergy := 23931.543050; stLENS2_428[531].fLow := 6.581560; stLENS2_428[531].fHigh := 17.389651;
    stLENS2_428[532].fEnergy := 23979.454031; stLENS2_428[532].fLow := 6.557006; stLENS2_428[532].fHigh := 17.310555;
    stLENS2_428[533].fEnergy := 24027.460930; stLENS2_428[533].fLow := 6.532543; stLENS2_428[533].fHigh := 17.231868;
    stLENS2_428[534].fEnergy := 24075.563939; stLENS2_428[534].fLow := 6.508172; stLENS2_428[534].fHigh := 17.153589;
    stLENS2_428[535].fEnergy := 24123.763250; stLENS2_428[535].fLow := 6.483892; stLENS2_428[535].fHigh := 17.075715;
    stLENS2_428[536].fEnergy := 24172.059056; stLENS2_428[536].fLow := 6.459703; stLENS2_428[536].fHigh := 16.998244;
    stLENS2_428[537].fEnergy := 24220.451551; stLENS2_428[537].fLow := 6.435603; stLENS2_428[537].fHigh := 16.921173;
    stLENS2_428[538].fEnergy := 24268.940927; stLENS2_428[538].fLow := 6.411594; stLENS2_428[538].fHigh := 16.844501;
    stLENS2_428[539].fEnergy := 24317.527379; stLENS2_428[539].fLow := 6.387674; stLENS2_428[539].fHigh := 16.768225;
    stLENS2_428[540].fEnergy := 24366.211101; stLENS2_428[540].fLow := 6.363843; stLENS2_428[540].fHigh := 16.692342;
    stLENS2_428[541].fEnergy := 24414.992288; stLENS2_428[541].fLow := 6.340102; stLENS2_428[541].fHigh := 16.616851;
    stLENS2_428[542].fEnergy := 24463.871136; stLENS2_428[542].fLow := 6.316449; stLENS2_428[542].fHigh := 16.541750;
    stLENS2_428[543].fEnergy := 24512.847838; stLENS2_428[543].fLow := 6.292884; stLENS2_428[543].fHigh := 16.467036;
    stLENS2_428[544].fEnergy := 24561.922592; stLENS2_428[544].fLow := 6.269407; stLENS2_428[544].fHigh := 16.392706;
    stLENS2_428[545].fEnergy := 24611.095594; stLENS2_428[545].fLow := 6.246017; stLENS2_428[545].fHigh := 16.318760;
    stLENS2_428[546].fEnergy := 24660.367040; stLENS2_428[546].fLow := 6.222715; stLENS2_428[546].fHigh := 16.245194;
    stLENS2_428[547].fEnergy := 24709.737128; stLENS2_428[547].fLow := 6.199500; stLENS2_428[547].fHigh := 16.172007;
    stLENS2_428[548].fEnergy := 24759.206055; stLENS2_428[548].fLow := 6.176372; stLENS2_428[548].fHigh := 16.099197;
    stLENS2_428[549].fEnergy := 24808.774018; stLENS2_428[549].fLow := 6.153329; stLENS2_428[549].fHigh := 16.026760;
    stLENS2_428[550].fEnergy := 24858.441217; stLENS2_428[550].fLow := 6.130373; stLENS2_428[550].fHigh := 15.954696;
    stLENS2_428[551].fEnergy := 24908.207849; stLENS2_428[551].fLow := 6.107502; stLENS2_428[551].fHigh := 15.883002;
    stLENS2_428[552].fEnergy := 24958.074115; stLENS2_428[552].fLow := 6.084717; stLENS2_428[552].fHigh := 15.811676;
    stLENS2_428[553].fEnergy := 25008.040212; stLENS2_428[553].fLow := 6.062017; stLENS2_428[553].fHigh := 15.740716;
    stLENS2_428[554].fEnergy := 25058.106342; stLENS2_428[554].fLow := 6.039401; stLENS2_428[554].fHigh := 15.670120;
    stLENS2_428[555].fEnergy := 25108.272705; stLENS2_428[555].fLow := 6.016870; stLENS2_428[555].fHigh := 15.599886;
    stLENS2_428[556].fEnergy := 25158.539500; stLENS2_428[556].fLow := 5.994422; stLENS2_428[556].fHigh := 15.530011;
    stLENS2_428[557].fEnergy := 25208.906930; stLENS2_428[557].fLow := 5.972059; stLENS2_428[557].fHigh := 15.460495;
    stLENS2_428[558].fEnergy := 25259.375195; stLENS2_428[558].fLow := 5.949779; stLENS2_428[558].fHigh := 15.391334;
    stLENS2_428[559].fEnergy := 25309.944498; stLENS2_428[559].fLow := 5.927582; stLENS2_428[559].fHigh := 15.322527;
    stLENS2_428[560].fEnergy := 25360.615041; stLENS2_428[560].fLow := 5.905468; stLENS2_428[560].fHigh := 15.254072;
    stLENS2_428[561].fEnergy := 25411.387026; stLENS2_428[561].fLow := 5.883436; stLENS2_428[561].fHigh := 15.185967;
    stLENS2_428[562].fEnergy := 25462.260656; stLENS2_428[562].fLow := 5.861487; stLENS2_428[562].fHigh := 15.118210;
    stLENS2_428[563].fEnergy := 25513.236136; stLENS2_428[563].fLow := 5.839619; stLENS2_428[563].fHigh := 15.050799;
    stLENS2_428[564].fEnergy := 25564.313669; stLENS2_428[564].fLow := 5.817833; stLENS2_428[564].fHigh := 14.983731;
    stLENS2_428[565].fEnergy := 25615.493459; stLENS2_428[565].fLow := 5.796128; stLENS2_428[565].fHigh := 14.917006;
    stLENS2_428[566].fEnergy := 25666.775711; stLENS2_428[566].fLow := 5.774505; stLENS2_428[566].fHigh := 14.850622;
    stLENS2_428[567].fEnergy := 25718.160630; stLENS2_428[567].fLow := 5.752962; stLENS2_428[567].fHigh := 14.784575;
    stLENS2_428[568].fEnergy := 25769.648422; stLENS2_428[568].fLow := 5.731499; stLENS2_428[568].fHigh := 14.718865;
    stLENS2_428[569].fEnergy := 25821.239293; stLENS2_428[569].fLow := 5.710116; stLENS2_428[569].fHigh := 14.653489;
    stLENS2_428[570].fEnergy := 25872.933448; stLENS2_428[570].fLow := 5.688814; stLENS2_428[570].fHigh := 14.588447;
    stLENS2_428[571].fEnergy := 25924.731096; stLENS2_428[571].fLow := 5.667590; stLENS2_428[571].fHigh := 14.523735;
    stLENS2_428[572].fEnergy := 25976.632442; stLENS2_428[572].fLow := 5.646446; stLENS2_428[572].fHigh := 14.459352;
    stLENS2_428[573].fEnergy := 26028.637695; stLENS2_428[573].fLow := 5.625381; stLENS2_428[573].fHigh := 14.395296;
    stLENS2_428[574].fEnergy := 26080.747062; stLENS2_428[574].fLow := 5.604394; stLENS2_428[574].fHigh := 14.331565;
    stLENS2_428[575].fEnergy := 26132.960752; stLENS2_428[575].fLow := 5.583486; stLENS2_428[575].fHigh := 14.268159;
    stLENS2_428[576].fEnergy := 26185.278975; stLENS2_428[576].fLow := 5.562655; stLENS2_428[576].fHigh := 14.205073;
    stLENS2_428[577].fEnergy := 26237.701938; stLENS2_428[577].fLow := 5.541903; stLENS2_428[577].fHigh := 14.142308;
    stLENS2_428[578].fEnergy := 26290.229852; stLENS2_428[578].fLow := 5.521227; stLENS2_428[578].fHigh := 14.079861;
    stLENS2_428[579].fEnergy := 26342.862928; stLENS2_428[579].fLow := 5.500629; stLENS2_428[579].fHigh := 14.017731;
    stLENS2_428[580].fEnergy := 26395.601374; stLENS2_428[580].fLow := 5.480108; stLENS2_428[580].fHigh := 13.955915;
    stLENS2_428[581].fEnergy := 26448.445404; stLENS2_428[581].fLow := 5.459663; stLENS2_428[581].fHigh := 13.894412;
    stLENS2_428[582].fEnergy := 26501.395226; stLENS2_428[582].fLow := 5.439295; stLENS2_428[582].fHigh := 13.833220;
    stLENS2_428[583].fEnergy := 26554.451055; stLENS2_428[583].fLow := 5.419002; stLENS2_428[583].fHigh := 13.772337;
    stLENS2_428[584].fEnergy := 26607.613102; stLENS2_428[584].fLow := 5.398786; stLENS2_428[584].fHigh := 13.711762;
    stLENS2_428[585].fEnergy := 26660.881578; stLENS2_428[585].fLow := 5.378644; stLENS2_428[585].fHigh := 13.651494;
    stLENS2_428[586].fEnergy := 26714.256699; stLENS2_428[586].fLow := 5.358578; stLENS2_428[586].fHigh := 13.591529;
    stLENS2_428[587].fEnergy := 26767.738676; stLENS2_428[587].fLow := 5.338587; stLENS2_428[587].fHigh := 13.531868;
    stLENS2_428[588].fEnergy := 26821.327725; stLENS2_428[588].fLow := 5.318670; stLENS2_428[588].fHigh := 13.472507;
    stLENS2_428[589].fEnergy := 26875.024059; stLENS2_428[589].fLow := 5.298827; stLENS2_428[589].fHigh := 13.413446;
    stLENS2_428[590].fEnergy := 26928.827893; stLENS2_428[590].fLow := 5.279059; stLENS2_428[590].fHigh := 13.354682;
    stLENS2_428[591].fEnergy := 26982.739442; stLENS2_428[591].fLow := 5.259364; stLENS2_428[591].fHigh := 13.296214;
    stLENS2_428[592].fEnergy := 27036.758923; stLENS2_428[592].fLow := 5.239743; stLENS2_428[592].fHigh := 13.238041;
    stLENS2_428[593].fEnergy := 27090.886550; stLENS2_428[593].fLow := 5.220195; stLENS2_428[593].fHigh := 13.180160;
    stLENS2_428[594].fEnergy := 27145.122541; stLENS2_428[594].fLow := 5.200720; stLENS2_428[594].fHigh := 13.122571;
    stLENS2_428[595].fEnergy := 27199.467113; stLENS2_428[595].fLow := 5.181318; stLENS2_428[595].fHigh := 13.065271;
    stLENS2_428[596].fEnergy := 27253.920482; stLENS2_428[596].fLow := 5.161988; stLENS2_428[596].fHigh := 13.008259;
    stLENS2_428[597].fEnergy := 27308.482867; stLENS2_428[597].fLow := 5.142730; stLENS2_428[597].fHigh := 12.951533;
    stLENS2_428[598].fEnergy := 27363.154486; stLENS2_428[598].fLow := 5.123544; stLENS2_428[598].fHigh := 12.895093;
    stLENS2_428[599].fEnergy := 27417.935558; stLENS2_428[599].fLow := 5.104429; stLENS2_428[599].fHigh := 12.838935;
    stLENS2_428[600].fEnergy := 27472.826302; stLENS2_428[600].fLow := 5.085386; stLENS2_428[600].fHigh := 12.783059;
    stLENS2_428[601].fEnergy := 27527.826937; stLENS2_428[601].fLow := 5.066414; stLENS2_428[601].fHigh := 12.727463;
    stLENS2_428[602].fEnergy := 27582.937683; stLENS2_428[602].fLow := 5.047513; stLENS2_428[602].fHigh := 12.672146;
    stLENS2_428[603].fEnergy := 27638.158761; stLENS2_428[603].fLow := 5.028682; stLENS2_428[603].fHigh := 12.617106;
    stLENS2_428[604].fEnergy := 27693.490392; stLENS2_428[604].fLow := 5.009921; stLENS2_428[604].fHigh := 12.562341;
    stLENS2_428[605].fEnergy := 27748.932796; stLENS2_428[605].fLow := 4.991231; stLENS2_428[605].fHigh := 12.507850;
    stLENS2_428[606].fEnergy := 27804.486197; stLENS2_428[606].fLow := 4.972610; stLENS2_428[606].fHigh := 12.453632;
    stLENS2_428[607].fEnergy := 27860.150815; stLENS2_428[607].fLow := 4.954058; stLENS2_428[607].fHigh := 12.399684;
    stLENS2_428[608].fEnergy := 27915.926874; stLENS2_428[608].fLow := 4.935576; stLENS2_428[608].fHigh := 12.346007;
    stLENS2_428[609].fEnergy := 27971.814597; stLENS2_428[609].fLow := 4.917163; stLENS2_428[609].fHigh := 12.292597;
    stLENS2_428[610].fEnergy := 28027.814207; stLENS2_428[610].fLow := 4.898818; stLENS2_428[610].fHigh := 12.239454;
    stLENS2_428[611].fEnergy := 28083.925929; stLENS2_428[611].fLow := 4.880542; stLENS2_428[611].fHigh := 12.186576;
    stLENS2_428[612].fEnergy := 28140.149986; stLENS2_428[612].fLow := 4.862334; stLENS2_428[612].fHigh := 12.133961;
    stLENS2_428[613].fEnergy := 28196.486604; stLENS2_428[613].fLow := 4.844194; stLENS2_428[613].fHigh := 12.081609;
    stLENS2_428[614].fEnergy := 28252.936008; stLENS2_428[614].fLow := 4.826122; stLENS2_428[614].fHigh := 12.029518;
    stLENS2_428[615].fEnergy := 28309.498423; stLENS2_428[615].fLow := 4.808117; stLENS2_428[615].fHigh := 11.977685;
    stLENS2_428[616].fEnergy := 28366.174077; stLENS2_428[616].fLow := 4.790179; stLENS2_428[616].fHigh := 11.926111;
    stLENS2_428[617].fEnergy := 28422.963195; stLENS2_428[617].fLow := 4.772309; stLENS2_428[617].fHigh := 11.874794;
    stLENS2_428[618].fEnergy := 28479.866005; stLENS2_428[618].fLow := 4.754504; stLENS2_428[618].fHigh := 11.823731;
    stLENS2_428[619].fEnergy := 28536.882735; stLENS2_428[619].fLow := 4.736767; stLENS2_428[619].fHigh := 11.772922;
    stLENS2_428[620].fEnergy := 28594.013612; stLENS2_428[620].fLow := 4.719095; stLENS2_428[620].fHigh := 11.722366;
    stLENS2_428[621].fEnergy := 28651.258866; stLENS2_428[621].fLow := 4.701490; stLENS2_428[621].fHigh := 11.672060;
    stLENS2_428[622].fEnergy := 28708.618724; stLENS2_428[622].fLow := 4.683950; stLENS2_428[622].fHigh := 11.622005;
    stLENS2_428[623].fEnergy := 28766.093417; stLENS2_428[623].fLow := 4.666475; stLENS2_428[623].fHigh := 11.572197;
    stLENS2_428[624].fEnergy := 28823.683175; stLENS2_428[624].fLow := 4.649066; stLENS2_428[624].fHigh := 11.522636;
    stLENS2_428[625].fEnergy := 28881.388227; stLENS2_428[625].fLow := 4.631722; stLENS2_428[625].fHigh := 11.473321;
    stLENS2_428[626].fEnergy := 28939.208804; stLENS2_428[626].fLow := 4.614442; stLENS2_428[626].fHigh := 11.424250;
    stLENS2_428[627].fEnergy := 28997.145139; stLENS2_428[627].fLow := 4.597227; stLENS2_428[627].fHigh := 11.375422;
    stLENS2_428[628].fEnergy := 29055.197462; stLENS2_428[628].fLow := 4.580076; stLENS2_428[628].fHigh := 11.326835;
    stLENS2_428[629].fEnergy := 29113.366006; stLENS2_428[629].fLow := 4.562989; stLENS2_428[629].fHigh := 11.278489;
    stLENS2_428[630].fEnergy := 29171.651004; stLENS2_428[630].fLow := 4.545966; stLENS2_428[630].fHigh := 11.230381;
    stLENS2_428[631].fEnergy := 29230.052688; stLENS2_428[631].fLow := 4.529006; stLENS2_428[631].fHigh := 11.182512;
    stLENS2_428[632].fEnergy := 29288.571293; stLENS2_428[632].fLow := 4.512109; stLENS2_428[632].fHigh := 11.134878;
    stLENS2_428[633].fEnergy := 29347.207052; stLENS2_428[633].fLow := 4.495276; stLENS2_428[633].fHigh := 11.087480;
    stLENS2_428[634].fEnergy := 29405.960199; stLENS2_428[634].fLow := 4.478505; stLENS2_428[634].fHigh := 11.040315;
    stLENS2_428[635].fEnergy := 29464.830971; stLENS2_428[635].fLow := 4.461797; stLENS2_428[635].fHigh := 10.993383;
    stLENS2_428[636].fEnergy := 29523.819602; stLENS2_428[636].fLow := 4.445152; stLENS2_428[636].fHigh := 10.946683;
    stLENS2_428[637].fEnergy := 29582.926328; stLENS2_428[637].fLow := 4.428568; stLENS2_428[637].fHigh := 10.900212;
    stLENS2_428[638].fEnergy := 29642.151386; stLENS2_428[638].fLow := 4.412046; stLENS2_428[638].fHigh := 10.853970;
    stLENS2_428[639].fEnergy := 29701.495012; stLENS2_428[639].fLow := 4.395586; stLENS2_428[639].fHigh := 10.807955;
    stLENS2_428[640].fEnergy := 29760.957445; stLENS2_428[640].fLow := 4.379188; stLENS2_428[640].fHigh := 10.762167;
    stLENS2_428[641].fEnergy := 29820.538922; stLENS2_428[641].fLow := 4.362850; stLENS2_428[641].fHigh := 10.716604;
    stLENS2_428[642].fEnergy := 29880.239680; stLENS2_428[642].fLow := 4.346574; stLENS2_428[642].fHigh := 10.671265;
    stLENS2_428[643].fEnergy := 29940.059960; stLENS2_428[643].fLow := 4.330358; stLENS2_428[643].fHigh := 10.626148;
    stLENS2_428[644].fEnergy := 30000.000000; stLENS2_428[644].fLow := 4.314202; stLENS2_428[644].fHigh := 10.581253;
    stLENS2_428[645].fEnergy := 30068.760232; stLENS2_428[645].fLow := 4.295783; stLENS2_428[645].fHigh := 10.529640;
    stLENS2_428[646].fEnergy := 30128.957930; stLENS2_428[646].fLow := 4.279757; stLENS2_428[646].fHigh := 10.485001;
    stLENS2_428[647].fEnergy := 30189.276144; stLENS2_428[647].fLow := 4.263791; stLENS2_428[647].fHigh := 10.440550;
    stLENS2_428[648].fEnergy := 30249.715115; stLENS2_428[648].fLow := 4.247884; stLENS2_428[648].fHigh := 10.396289;
    stLENS2_428[649].fEnergy := 30310.275085; stLENS2_428[649].fLow := 4.232036; stLENS2_428[649].fHigh := 10.352214;
    stLENS2_428[650].fEnergy := 30370.956297; stLENS2_428[650].fLow := 4.216247; stLENS2_428[650].fHigh := 10.308327;
    stLENS2_428[651].fEnergy := 30431.758992; stLENS2_428[651].fLow := 4.200518; stLENS2_428[651].fHigh := 10.264626;
    stLENS2_428[652].fEnergy := 30492.683414; stLENS2_428[652].fLow := 4.184847; stLENS2_428[652].fHigh := 10.221110;
    stLENS2_428[653].fEnergy := 30553.729807; stLENS2_428[653].fLow := 4.169234; stLENS2_428[653].fHigh := 10.177778;
    stLENS2_428[654].fEnergy := 30614.898414; stLENS2_428[654].fLow := 4.153680; stLENS2_428[654].fHigh := 10.134631;
    stLENS2_428[655].fEnergy := 30676.189482; stLENS2_428[655].fLow := 4.138184; stLENS2_428[655].fHigh := 10.091666;
    stLENS2_428[656].fEnergy := 30737.603254; stLENS2_428[656].fLow := 4.122745; stLENS2_428[656].fHigh := 10.048883;
    stLENS2_428[657].fEnergy := 30799.139977; stLENS2_428[657].fLow := 4.107365; stLENS2_428[657].fHigh := 10.006282;
    stLENS2_428[658].fEnergy := 30860.799896; stLENS2_428[658].fLow := 4.092041; stLENS2_428[658].fHigh := 9.963861;
    stLENS2_428[659].fEnergy := 30922.583259; stLENS2_428[659].fLow := 4.076775; stLENS2_428[659].fHigh := 9.921620;
    stLENS2_428[660].fEnergy := 30984.490312; stLENS2_428[660].fLow := 4.061566; stLENS2_428[660].fHigh := 9.879558;
    stLENS2_428[661].fEnergy := 31046.521303; stLENS2_428[661].fLow := 4.046413; stLENS2_428[661].fHigh := 9.837675;
    stLENS2_428[662].fEnergy := 31108.676480; stLENS2_428[662].fLow := 4.031317; stLENS2_428[662].fHigh := 9.795969;
    stLENS2_428[663].fEnergy := 31170.956091; stLENS2_428[663].fLow := 4.016277; stLENS2_428[663].fHigh := 9.754440;
    stLENS2_428[664].fEnergy := 31233.360387; stLENS2_428[664].fLow := 4.001294; stLENS2_428[664].fHigh := 9.713086;
    stLENS2_428[665].fEnergy := 31295.889616; stLENS2_428[665].fLow := 3.986366; stLENS2_428[665].fHigh := 9.671909;
    stLENS2_428[666].fEnergy := 31358.544029; stLENS2_428[666].fLow := 3.971494; stLENS2_428[666].fHigh := 9.630906;
    stLENS2_428[667].fEnergy := 31421.323876; stLENS2_428[667].fLow := 3.956678; stLENS2_428[667].fHigh := 9.590076;
    stLENS2_428[668].fEnergy := 31484.229408; stLENS2_428[668].fLow := 3.941916; stLENS2_428[668].fHigh := 9.549420;
    stLENS2_428[669].fEnergy := 31547.260878; stLENS2_428[669].fLow := 3.927210; stLENS2_428[669].fHigh := 9.508936;
    stLENS2_428[670].fEnergy := 31610.418536; stLENS2_428[670].fLow := 3.912559; stLENS2_428[670].fHigh := 9.468624;
    stLENS2_428[671].fEnergy := 31673.702636; stLENS2_428[671].fLow := 3.897962; stLENS2_428[671].fHigh := 9.428482;
    stLENS2_428[672].fEnergy := 31737.113431; stLENS2_428[672].fLow := 3.883420; stLENS2_428[672].fHigh := 9.388511;
    stLENS2_428[673].fEnergy := 31800.651174; stLENS2_428[673].fLow := 3.868932; stLENS2_428[673].fHigh := 9.348709;
    stLENS2_428[674].fEnergy := 31864.316120; stLENS2_428[674].fLow := 3.854498; stLENS2_428[674].fHigh := 9.309076;
    stLENS2_428[675].fEnergy := 31928.108524; stLENS2_428[675].fLow := 3.840118; stLENS2_428[675].fHigh := 9.269611;
    stLENS2_428[676].fEnergy := 31992.028640; stLENS2_428[676].fLow := 3.825792; stLENS2_428[676].fHigh := 9.230314;
    stLENS2_428[677].fEnergy := 32056.076724; stLENS2_428[677].fLow := 3.811519; stLENS2_428[677].fHigh := 9.191182;
    stLENS2_428[678].fEnergy := 32120.253032; stLENS2_428[678].fLow := 3.797299; stLENS2_428[678].fHigh := 9.152217;
    stLENS2_428[679].fEnergy := 32184.557822; stLENS2_428[679].fLow := 3.783133; stLENS2_428[679].fHigh := 9.113417;
    stLENS2_428[680].fEnergy := 32248.991349; stLENS2_428[680].fLow := 3.769019; stLENS2_428[680].fHigh := 9.074782;
    stLENS2_428[681].fEnergy := 32313.553873; stLENS2_428[681].fLow := 3.754958; stLENS2_428[681].fHigh := 9.036310;
    stLENS2_428[682].fEnergy := 32378.245651; stLENS2_428[682].fLow := 3.740949; stLENS2_428[682].fHigh := 8.998001;
    stLENS2_428[683].fEnergy := 32443.066942; stLENS2_428[683].fLow := 3.726993; stLENS2_428[683].fHigh := 8.959855;
    stLENS2_428[684].fEnergy := 32508.018005; stLENS2_428[684].fLow := 3.713088; stLENS2_428[684].fHigh := 8.921871;
    stLENS2_428[685].fEnergy := 32573.099101; stLENS2_428[685].fLow := 3.699236; stLENS2_428[685].fHigh := 8.884047;
    stLENS2_428[686].fEnergy := 32638.310488; stLENS2_428[686].fLow := 3.685435; stLENS2_428[686].fHigh := 8.846384;
    stLENS2_428[687].fEnergy := 32703.652430; stLENS2_428[687].fLow := 3.671686; stLENS2_428[687].fHigh := 8.808880;
    stLENS2_428[688].fEnergy := 32769.125185; stLENS2_428[688].fLow := 3.657988; stLENS2_428[688].fHigh := 8.771536;
    stLENS2_428[689].fEnergy := 32834.729018; stLENS2_428[689].fLow := 3.644341; stLENS2_428[689].fHigh := 8.734350;
    stLENS2_428[690].fEnergy := 32900.464189; stLENS2_428[690].fLow := 3.630745; stLENS2_428[690].fHigh := 8.697321;
    stLENS2_428[691].fEnergy := 32966.330962; stLENS2_428[691].fLow := 3.617199; stLENS2_428[691].fHigh := 8.660450;
    stLENS2_428[692].fEnergy := 33032.329601; stLENS2_428[692].fLow := 3.603705; stLENS2_428[692].fHigh := 8.623735;
    stLENS2_428[693].fEnergy := 33098.460369; stLENS2_428[693].fLow := 3.590260; stLENS2_428[693].fHigh := 8.587175;
    stLENS2_428[694].fEnergy := 33164.723530; stLENS2_428[694].fLow := 3.576866; stLENS2_428[694].fHigh := 8.550770;
    stLENS2_428[695].fEnergy := 33231.119351; stLENS2_428[695].fLow := 3.563522; stLENS2_428[695].fHigh := 8.514520;
    stLENS2_428[696].fEnergy := 33297.648096; stLENS2_428[696].fLow := 3.550227; stLENS2_428[696].fHigh := 8.478424;
    stLENS2_428[697].fEnergy := 33364.310032; stLENS2_428[697].fLow := 3.536982; stLENS2_428[697].fHigh := 8.442480;
    stLENS2_428[698].fEnergy := 33431.105426; stLENS2_428[698].fLow := 3.523787; stLENS2_428[698].fHigh := 8.406689;
    stLENS2_428[699].fEnergy := 33498.034543; stLENS2_428[699].fLow := 3.510641; stLENS2_428[699].fHigh := 8.371050;
    stLENS2_428[700].fEnergy := 33565.097653; stLENS2_428[700].fLow := 3.497543; stLENS2_428[700].fHigh := 8.335561;
    stLENS2_428[701].fEnergy := 33632.295023; stLENS2_428[701].fLow := 3.484495; stLENS2_428[701].fHigh := 8.300223;
    stLENS2_428[702].fEnergy := 33699.626923; stLENS2_428[702].fLow := 3.471495; stLENS2_428[702].fHigh := 8.265035;
    stLENS2_428[703].fEnergy := 33767.093621; stLENS2_428[703].fLow := 3.458544; stLENS2_428[703].fHigh := 8.229996;
    stLENS2_428[704].fEnergy := 33834.695387; stLENS2_428[704].fLow := 3.445641; stLENS2_428[704].fHigh := 8.195106;
    stLENS2_428[705].fEnergy := 33902.432493; stLENS2_428[705].fLow := 3.432787; stLENS2_428[705].fHigh := 8.160364;
    stLENS2_428[706].fEnergy := 33970.305208; stLENS2_428[706].fLow := 3.419980; stLENS2_428[706].fHigh := 8.125768;
    stLENS2_428[707].fEnergy := 34038.313804; stLENS2_428[707].fLow := 3.407221; stLENS2_428[707].fHigh := 8.091320;
    stLENS2_428[708].fEnergy := 34106.458554; stLENS2_428[708].fLow := 3.394510; stLENS2_428[708].fHigh := 8.057018;
    stLENS2_428[709].fEnergy := 34174.739729; stLENS2_428[709].fLow := 3.381846; stLENS2_428[709].fHigh := 8.022861;
    stLENS2_428[710].fEnergy := 34243.157604; stLENS2_428[710].fLow := 3.369229; stLENS2_428[710].fHigh := 7.988848;
    stLENS2_428[711].fEnergy := 34311.712451; stLENS2_428[711].fLow := 3.356659; stLENS2_428[711].fHigh := 7.954980;
    stLENS2_428[712].fEnergy := 34380.404545; stLENS2_428[712].fLow := 3.344137; stLENS2_428[712].fHigh := 7.921256;
    stLENS2_428[713].fEnergy := 34449.234161; stLENS2_428[713].fLow := 3.331660; stLENS2_428[713].fHigh := 7.887674;
    stLENS2_428[714].fEnergy := 34518.201574; stLENS2_428[714].fLow := 3.319231; stLENS2_428[714].fHigh := 7.854235;
    stLENS2_428[715].fEnergy := 34587.307059; stLENS2_428[715].fLow := 3.306848; stLENS2_428[715].fHigh := 7.820938;
    stLENS2_428[716].fEnergy := 34656.550894; stLENS2_428[716].fLow := 3.294511; stLENS2_428[716].fHigh := 7.787782;
    stLENS2_428[717].fEnergy := 34725.933355; stLENS2_428[717].fLow := 3.282220; stLENS2_428[717].fHigh := 7.754766;
    stLENS2_428[718].fEnergy := 34795.454720; stLENS2_428[718].fLow := 3.269975; stLENS2_428[718].fHigh := 7.721891;
    stLENS2_428[719].fEnergy := 34865.115267; stLENS2_428[719].fLow := 3.257776; stLENS2_428[719].fHigh := 7.689154;
    stLENS2_428[720].fEnergy := 34934.915274; stLENS2_428[720].fLow := 3.245622; stLENS2_428[720].fHigh := 7.656557;
    stLENS2_428[721].fEnergy := 35004.855021; stLENS2_428[721].fLow := 3.233513; stLENS2_428[721].fHigh := 7.624097;
    stLENS2_428[722].fEnergy := 35074.934788; stLENS2_428[722].fLow := 3.221450; stLENS2_428[722].fHigh := 7.591776;
    stLENS2_428[723].fEnergy := 35145.154854; stLENS2_428[723].fLow := 3.209432; stLENS2_428[723].fHigh := 7.559591;
    stLENS2_428[724].fEnergy := 35215.515501; stLENS2_428[724].fLow := 3.197458; stLENS2_428[724].fHigh := 7.527543;
    stLENS2_428[725].fEnergy := 35286.017010; stLENS2_428[725].fLow := 3.185529; stLENS2_428[725].fHigh := 7.495631;
    stLENS2_428[726].fEnergy := 35356.659663; stLENS2_428[726].fLow := 3.173645; stLENS2_428[726].fHigh := 7.463853;
    stLENS2_428[727].fEnergy := 35427.443743; stLENS2_428[727].fLow := 3.161805; stLENS2_428[727].fHigh := 7.432211;
    stLENS2_428[728].fEnergy := 35498.369532; stLENS2_428[728].fLow := 3.150009; stLENS2_428[728].fHigh := 7.400703;
    stLENS2_428[729].fEnergy := 35569.437315; stLENS2_428[729].fLow := 3.138258; stLENS2_428[729].fHigh := 7.369328;
    stLENS2_428[730].fEnergy := 35640.647376; stLENS2_428[730].fLow := 3.126550; stLENS2_428[730].fHigh := 7.338087;
    stLENS2_428[731].fEnergy := 35712.000000; stLENS2_428[731].fLow := 3.114885; stLENS2_428[731].fHigh := 7.306977;
    stLENS2_428[732].fEnergy := 35783.495472; stLENS2_428[732].fLow := 3.103265; stLENS2_428[732].fHigh := 7.276000;
    stLENS2_428[733].fEnergy := 35855.134077; stLENS2_428[733].fLow := 3.091687; stLENS2_428[733].fHigh := 7.245154;
    stLENS2_428[734].fEnergy := 35926.916104; stLENS2_428[734].fLow := 3.080153; stLENS2_428[734].fHigh := 7.214439;


